// TIA Portal V20 export
FUNCTION_BLOCK "CallEquipment"   // FB25, LAD
TITLE = CallEquipment
// Template of an equipment module. This block contains the logic and futher calls (e.g. sequences, control modules, diagnostics etc.) of the equipment module.
// It can be used out of the box but also adapted to your own needs.
// stored: IsIECCheckEnabled true, MemoryReserve 100, Namespace Unit1.Em6, SetENOAutomatically true
   VAR_INPUT
      ZoneOperationEnable { ExternalWritable := 'False'} : "LWONIK_typeSafetyZoneManualOperation";
      unitEnableControlInterfaces { ExternalWritable := 'False'} : "LAF_typeEnableControlInterfaces";
      commandExcute { ExternalWritable := 'False'} : Bool;
   END_VAR
   VAR_IN_OUT
      unitStatus : "LAF_typeUnitStatus";   // Current unit status o be used in this EM
      emFeedback : "LUC_typeEmFeedback";   // Feedback of the EM to the Unit
      unitAlarmDB : "LAF_typeAlarms";   // Summarized EM Alarms for the Unit
   END_VAR
   VAR
      instSequenceVisionUnit { ExternalWritable := 'False'} : "Unit1.Em6.Sequence_1_VisionUnit";
      instSequenceVisionController { ExternalWritable := 'False'} : "Unit1.Em6.Sequence_2_VisionController";
      instSequenceQrRead { ExternalWritable := 'False'} : "Unit1.Em6.Sequence_3_QrRead";
      instVisionUnitInitializedJob1 { ExternalWritable := 'False'} : "LAF_SelectJob";
      instVisionUnitVisionPosJob2 { ExternalWritable := 'False'} : "LAF_SelectJob";
      instVisionUnitHomePosJob3 { ExternalWritable := 'False'} : "LAF_SelectJob";
      instVisionFullAutoJob10 { ExternalWritable := 'False'} : "LAF_SelectJob";
      instVisionControllerInitializedJob1 { ExternalWritable := 'False'} : "LAF_SelectJob";
      instVisionControllerInspectionJob2 { ExternalWritable := 'False'} : "LAF_SelectJob";
      instQrReaderInitializedJob1 { ExternalWritable := 'False'} : "LAF_SelectJob";
      instQrReaderQrReadJob2 { ExternalWritable := 'False'} : "LAF_SelectJob";
      instCmVisionAxisZ { ExternalWritable := 'False'} : "LBC_Axis64Pos_TecPlcCn";
      instCmVisionPusherSupportUpDown { ExternalWritable := 'False'} : "LBC_TwoWayActuatorCn";
      instCmVisionTriggerSensor { ExternalWritable := 'False'} : "LBC_DigitalSignalCn";
      instCmQrReader { ExternalWritable := 'False'} : "LER_QRread_SRX300";
      instCmQrReadHandy { ExternalWritable := 'False'} : "LER_QRread_DM8700";
      instVision_XGX2000 { ExternalWritable := 'False'} : "LER_Vision_XGX2000";
      instVision_XGX2000_Conversion { ExternalWritable := 'False'} : "LER_Vision_XGX2000_Conversion";
      instVisionAxisZControlInterlockSummary { ExternalWritable := 'False'} : "LER_Axis64Pos_InterlockSummary";
      instServoTorqueCal_DR9 { ExternalWritable := 'False'} : "LER_ServoTorqueCal";
      instLDrv701ControlVisionAxisZ { ExternalWritable := 'False'} : "LDrvSafe_SinaTlg701Control";   // Drive Telegram Function Library
      instLDrv701StatusVisionAxisZ { ExternalWritable := 'False'} : "LDrvSafe_SinaTlg701Status";   // Drive Telegram Function Library
      statUnitStatus { ExternalWritable := 'False'} : "LAF_typeUnitStatus";   // Unit Status used in this EM
      statAllBrakeTest { ExternalWritable := 'False'} : "LER_typeBrakeTestUnitCommands";
      instManageAlarms { ExternalWritable := 'False'} : "LAF_ManageAlarms";
      instEventsPFE { S7_SetPoint := 'True'} : "Unit1.Em6.EventsPFE";
      statPulse { ExternalWritable := 'False'} : Array[0..99] of Bool;
      statTonTimer { ExternalWritable := 'False'} : Array[0..99] of TON_TIME;
      statTofTimer { ExternalWritable := 'False'} : Array[0..99] of TOF_TIME;
      statEnableManualCmds { ExternalWritable := 'False'} : Bool;
      statGaugeCheck { ExternalWritable := 'False'} : Struct
         Type1Complete : Bool;
         Type3Compete : Bool;
      END_STRUCT;
      statSafeStateCheck { ExternalWritable := 'False'} : Struct
         VisionUnit : Bool;
         VisionController : Bool;
         VisionQrReader : Bool;
      END_STRUCT;
      statBobinID : String[32];
      citi_Ptrig : Array[0..20] of Bool;
      citiTon : Array[0..20] of TON_TIME;
      citi : Time;
      citiTest : Array[0..20] of Bool;
      statDataIncrease : Int;
   END_VAR
   VAR_TEMP
      tempScInProduction : Bool;   // Mode Production and StateComplete
      tempScNoProduction : Bool;   // Mode Manual and StateComplete
   END_VAR
   VAR CONSTANT
      TO_DO_INSERT_PRECONDITIONS_HERE : Bool := TRUE;   // Template : Add em specific conditions here
      NO_JOB : DInt;   // No job
      TRUE : Bool := TRUE;
      FALSE : Bool := FALSE;
      INIT_POSITION_NUMBER : SInt := -1;
      MIN_POSITION_NUMBER : SInt;
   END_VAR
   VAR_TEMP   // added for the SCL form of the ladder/FBD networks
      _w1 : Bool;
      _w2 : Bool;
      _w3 : Bool;
      _w4 : Bool;
      _w5 : Bool;
      _w6 : Bool;
      _w7 : Bool;
      _w8 : Bool;
      _w9 : Bool;
      _w10 : Bool;
      _w11 : Bool;
      _w12 : Bool;
      _w13 : Bool;
      _w14 : Bool;
      _w15 : Bool;
   END_VAR
BEGIN

REGION Network 1: BLOCK INFO HEADER
   // (company) / (C) Copyright (year)
   // ---------------------------------------------------------------------------------
   // Title:                             (Title of this block)
   // Comment/Function: (that is implemented in the block)
   // Library/Family:           (that the source is dedicated to)
   // Author:                        (department / person in charge / contact)
   // Target System:          (test system with FW version)
   // Engineering:              TIA Portal (SW version)
   // Restrictions:               (OB types, etc.)
   // Requirements:           (hardware, technological package, etc.)
   // ---------------------------------------------------------------------------------
   // Change log table:
   // Version          | Date             | Signature      | Expert in charge  | Changes applied ------------------------|----------------------|-------------------------|--------------------------------|-----------------------
   // 001.000.000 | yyyy-mm-dd | 0x00000000 | (name of expert) | First released version
END_REGION

REGION Network 2: DESCRIPTION
   // This is a template block provided by the Automation Framework. It can be used to create an own project.
   // The Block Info Header is prepared to put in your own data.
   // Description of the block could be added here and the docu created by Code2Docu.
END_REGION

REGION Network 3: ******************** Unit Input ********************
END_REGION

REGION Network 4: Em Nodes Brake Test
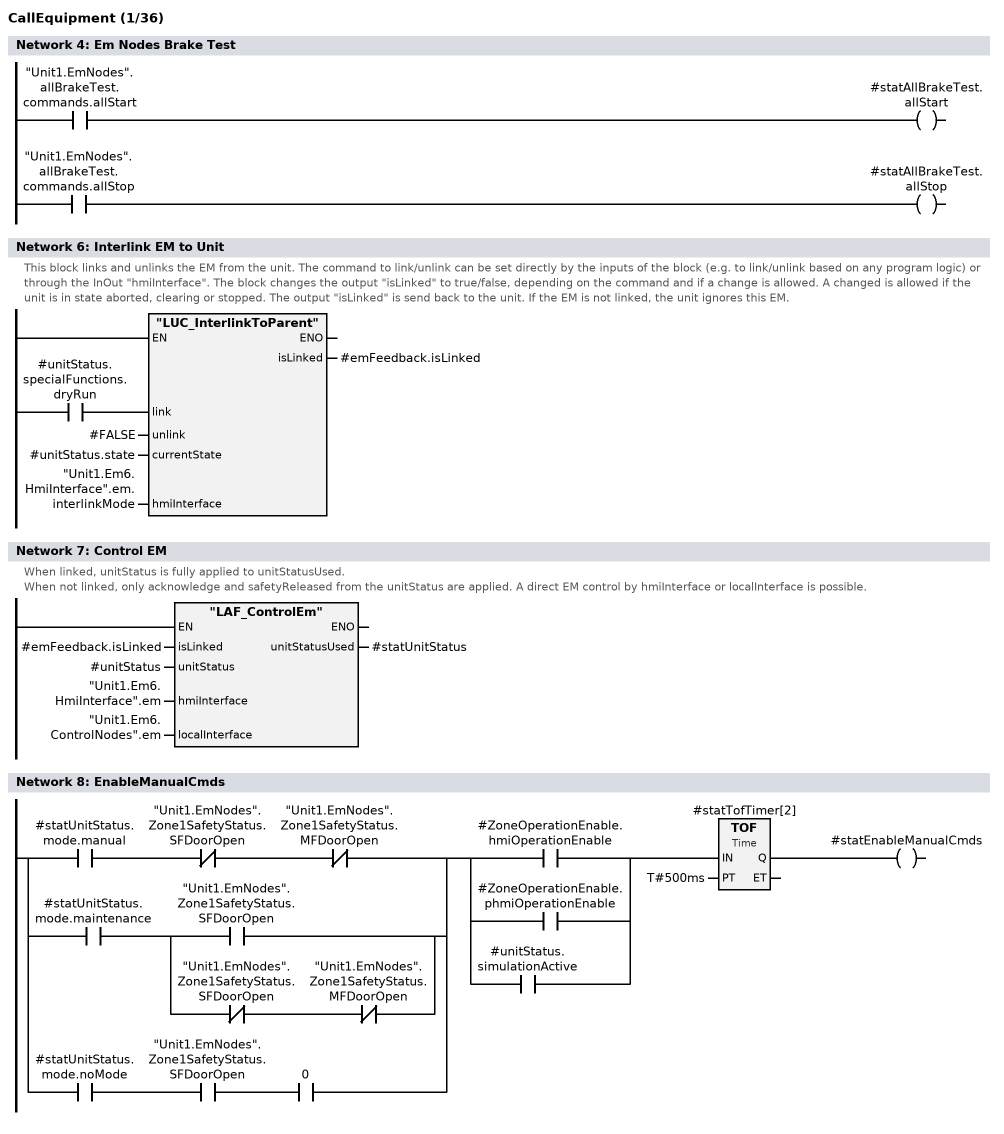
   RUNG wire#powerrail
      Contact( "Unit1.EmNodes".allBrakeTest.commands.allStart )
      Coil( #statAllBrakeTest.allStart )
   END_RUNG
   RUNG wire#powerrail
      Contact( "Unit1.EmNodes".allBrakeTest.commands.allStop )
      Coil( #statAllBrakeTest.allStop )
   END_RUNG
   // the same network as SCL:
   #statAllBrakeTest.allStart := "Unit1.EmNodes".allBrakeTest.commands.allStart;
   #statAllBrakeTest.allStop := "Unit1.EmNodes".allBrakeTest.commands.allStop;
END_REGION

REGION Network 5: ******************** Equipment Control ********************
END_REGION

REGION Network 6: Interlink EM to Unit
   // This block links and unlinks the EM from the unit. The command to link/unlink can be set directly by the inputs of the block (e.g. to link/unlink based on any program logic) or through the InOut "hmiInterface". The block changes the output "isLinked" to true/false, depending on the command and if a change is allowed. A changed is allowed if the unit is in state aborted, clearing or stopped. The output "isLinked" is send back to the unit. If the EM is not linked, the unit ignores this EM.
   RUNG wire#powerrail
      "LUC_InterlinkToParent"(link := wire#w1, unlink := #FALSE, currentState := #unitStatus.state, hmiInterface := "Unit1.Em6.HmiInterface".em.interlinkMode, isLinked => #emFeedback.isLinked)
   END_RUNG
   RUNG wire#powerrail
      Contact( #unitStatus.specialFunctions.dryRun )
   END_RUNG wire#w1
   // the same network as SCL:
   "LUC_InterlinkToParent"(link := #unitStatus.specialFunctions.dryRun,
                           unlink := #FALSE,
                           currentState := #unitStatus.state,
                           hmiInterface := "Unit1.Em6.HmiInterface".em.interlinkMode,
                           isLinked => #emFeedback.isLinked);
END_REGION

REGION Network 7: Control EM
   // When linked, unitStatus is fully applied to unitStatusUsed.
   // When not linked, only acknowledge and safetyReleased from the unitStatus are applied. A direct EM control by hmiInterface or localInterface is possible.
   RUNG wire#powerrail
      "LAF_ControlEm"(isLinked := #emFeedback.isLinked, unitStatus := #unitStatus, hmiInterface := "Unit1.Em6.HmiInterface".em, localInterface := "Unit1.Em6.ControlNodes".em, unitStatusUsed => #statUnitStatus)
   END_RUNG
   // the same network as SCL:
   "LAF_ControlEm"(isLinked := #emFeedback.isLinked,
                   unitStatus := #unitStatus,
                   hmiInterface := "Unit1.Em6.HmiInterface".em,
                   localInterface := "Unit1.Em6.ControlNodes".em,
                   unitStatusUsed => #statUnitStatus);
END_REGION

REGION Network 8: EnableManualCmds
   RUNG wire#powerrail
      Contact( #statUnitStatus.mode.manual )
      I_Contact( "Unit1.EmNodes".Zone1SafetyStatus.SFDoorOpen )
      I_Contact( "Unit1.EmNodes".Zone1SafetyStatus.MFDoorOpen )
      wire#w1
      Contact( #ZoneOperationEnable.hmiOperationEnable )
      wire#w3
      { S7_Templates := "time_type := Time" } #statTofTimer[2].TOF(pt := T#500ms, et =>)
      Coil( #statEnableManualCmds )
   END_RUNG
   RUNG wire#powerrail
      Contact( #statUnitStatus.mode.maintenance )
      wire#w2
      Contact( "Unit1.EmNodes".Zone1SafetyStatus.SFDoorOpen )
   END_RUNG wire#w1
   RUNG wire#w2
      I_Contact( "Unit1.EmNodes".Zone1SafetyStatus.SFDoorOpen )
      I_Contact( "Unit1.EmNodes".Zone1SafetyStatus.MFDoorOpen )
   END_RUNG wire#w1
   RUNG wire#powerrail
      Contact( #statUnitStatus.mode.noMode )
      Contact( "Unit1.EmNodes".Zone1SafetyStatus.SFDoorOpen )
      Contact( 0 )
   END_RUNG wire#w1
   RUNG wire#w1
      Contact( #ZoneOperationEnable.phmiOperationEnable )
   END_RUNG wire#w3
   RUNG wire#w1
      Contact( #unitStatus.simulationActive )
   END_RUNG wire#w3
   // the same network as SCL:
   #statTofTimer[2].TOF(IN := ((#statUnitStatus.mode.manual AND NOT "Unit1.EmNodes".Zone1SafetyStatus.SFDoorOpen AND NOT "Unit1.EmNodes".Zone1SafetyStatus.MFDoorOpen) OR (#statUnitStatus.mode.maintenance AND ("Unit1.EmNodes".Zone1SafetyStatus.SFDoorOpen OR (NOT "Unit1.EmNodes".Zone1SafetyStatus.SFDoorOpen AND NOT "Unit1.EmNodes".Zone1SafetyStatus.MFDoorOpen))) OR (#statUnitStatus.mode.noMode AND "Unit1.EmNodes".Zone1SafetyStatus.SFDoorOpen AND 0)) AND (#ZoneOperationEnable.hmiOperationEnable OR #ZoneOperationEnable.phmiOperationEnable OR #unitStatus.simulationActive),
                        PT := T#500ms);
   #statEnableManualCmds := #statTofTimer[2].Q;
END_REGION

REGION Network 9: Alarms Disabled
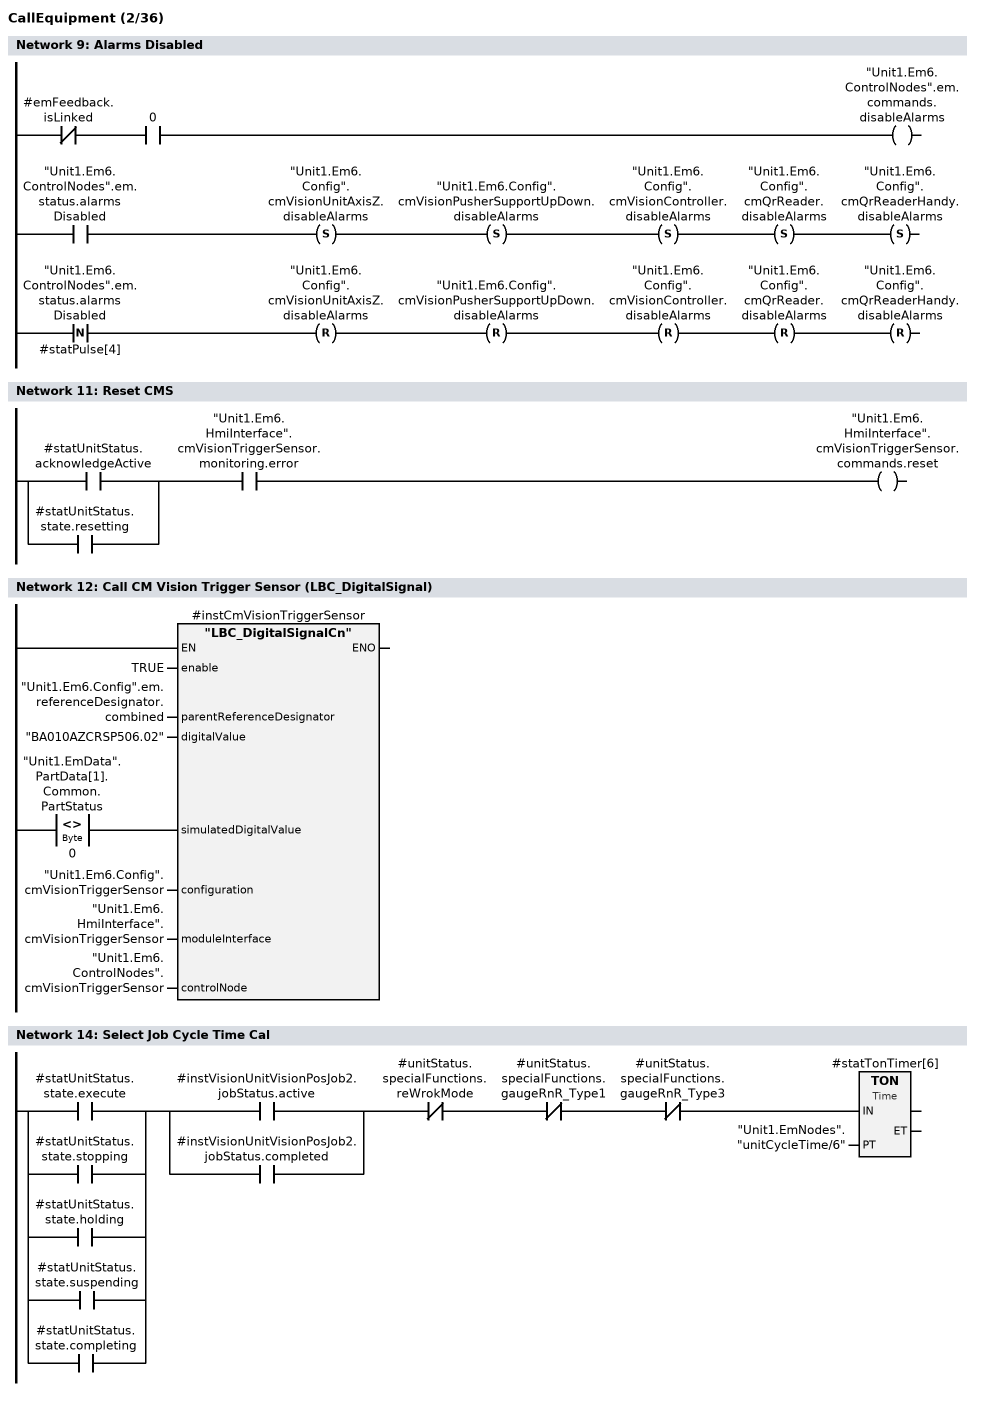
   RUNG wire#powerrail
      I_Contact( #emFeedback.isLinked )
      Contact( 0 )
      Coil( "Unit1.Em6.ControlNodes".em.commands.disableAlarms )
   END_RUNG
   RUNG wire#powerrail
      Contact( "Unit1.Em6.ControlNodes".em.status.alarmsDisabled )
      S_Coil( "Unit1.Em6.Config".cmVisionUnitAxisZ.disableAlarms )
      S_Coil( "Unit1.Em6.Config".cmVisionPusherSupportUpDown.disableAlarms )
      S_Coil( "Unit1.Em6.Config".cmVisionController.disableAlarms )
      S_Coil( "Unit1.Em6.Config".cmQrReader.disableAlarms )
      S_Coil( "Unit1.Em6.Config".cmQrReaderHandy.disableAlarms )
   END_RUNG
   RUNG wire#powerrail
      N_Contact(operand := "Unit1.Em6.ControlNodes".em.status.alarmsDisabled, bit := #statPulse[4])
      R_Coil( "Unit1.Em6.Config".cmVisionUnitAxisZ.disableAlarms )
      R_Coil( "Unit1.Em6.Config".cmVisionPusherSupportUpDown.disableAlarms )
      R_Coil( "Unit1.Em6.Config".cmVisionController.disableAlarms )
      R_Coil( "Unit1.Em6.Config".cmQrReader.disableAlarms )
      R_Coil( "Unit1.Em6.Config".cmQrReaderHandy.disableAlarms )
   END_RUNG
   // the same network as SCL:
   "Unit1.Em6.ControlNodes".em.commands.disableAlarms := NOT #emFeedback.isLinked AND 0;
   IF "Unit1.Em6.ControlNodes".em.status.alarmsDisabled THEN
       "Unit1.Em6.Config".cmVisionUnitAxisZ.disableAlarms := TRUE;
       "Unit1.Em6.Config".cmVisionPusherSupportUpDown.disableAlarms := TRUE;
       "Unit1.Em6.Config".cmVisionController.disableAlarms := TRUE;
       "Unit1.Em6.Config".cmQrReader.disableAlarms := TRUE;
       "Unit1.Em6.Config".cmQrReaderHandy.disableAlarms := TRUE;
   END_IF;
   #_w1 := NOT "Unit1.Em6.ControlNodes".em.status.alarmsDisabled AND #statPulse[4];   // falling edge of "Unit1.Em6.ControlNodes".em.status.alarmsDisabled
   #statPulse[4] := "Unit1.Em6.ControlNodes".em.status.alarmsDisabled;
   IF #_w1 THEN
       "Unit1.Em6.Config".cmVisionUnitAxisZ.disableAlarms := FALSE;
       "Unit1.Em6.Config".cmVisionPusherSupportUpDown.disableAlarms := FALSE;
       "Unit1.Em6.Config".cmVisionController.disableAlarms := FALSE;
       "Unit1.Em6.Config".cmQrReader.disableAlarms := FALSE;
       "Unit1.Em6.Config".cmQrReaderHandy.disableAlarms := FALSE;
   END_IF;
END_REGION

REGION Network 10: ******************** Control Modules (Sensors) ********************
   // Call control modules that are sensors before the em logic (jobs and sequence), so that the latest value is used in the logic.
END_REGION

REGION Network 11: Reset CMS
   RUNG wire#powerrail
      Contact( #statUnitStatus.acknowledgeActive )
      wire#w1
      Contact( "Unit1.Em6.HmiInterface".cmVisionTriggerSensor.monitoring.error )
      Coil( "Unit1.Em6.HmiInterface".cmVisionTriggerSensor.commands.reset )
   END_RUNG
   RUNG wire#powerrail
      Contact( #statUnitStatus.state.resetting )
   END_RUNG wire#w1
   // the same network as SCL:
   "Unit1.Em6.HmiInterface".cmVisionTriggerSensor.commands.reset := (#statUnitStatus.acknowledgeActive OR #statUnitStatus.state.resetting) AND "Unit1.Em6.HmiInterface".cmVisionTriggerSensor.monitoring.error;
END_REGION

REGION Network 12: Call CM Vision Trigger Sensor (LBC_DigitalSignal)
   RUNG wire#powerrail
      #instCmVisionTriggerSensor(simulatedDigitalValue := wire#w1, enable := TRUE, parentReferenceDesignator := "Unit1.Em6.Config".em.referenceDesignator.combined, digitalValue := "BA010AZCRSP506.02", configuration := "Unit1.Em6.Config".cmVisionTriggerSensor, moduleInterface := "Unit1.Em6.HmiInterface".cmVisionTriggerSensor, controlNode := "Unit1.Em6.ControlNodes".cmVisionTriggerSensor)
   END_RUNG
   RUNG wire#powerrail
      { S7_Templates := "SrcType := Byte" } NE_Contact(in1 := "Unit1.EmData".PartData[1].Common.PartStatus, in2 := 0)
   END_RUNG wire#w1
   // the same network as SCL:
   #instCmVisionTriggerSensor(enable := TRUE,   // "LBC_DigitalSignalCn"
                           parentReferenceDesignator := "Unit1.Em6.Config".em.referenceDesignator.combined,
                           digitalValue := "BA010AZCRSP506.02",
                           simulatedDigitalValue := "Unit1.EmData".PartData[1].Common.PartStatus <> 0,
                           configuration := "Unit1.Em6.Config".cmVisionTriggerSensor,
                           moduleInterface := "Unit1.Em6.HmiInterface".cmVisionTriggerSensor,
                           controlNode := "Unit1.Em6.ControlNodes".cmVisionTriggerSensor);
END_REGION

REGION Network 13: ******************** Equipment Logic ********************
END_REGION

REGION Network 14: Select Job Cycle Time Cal
   RUNG wire#powerrail
      Contact( #statUnitStatus.state.execute )
      wire#w1
      Contact( #instVisionUnitVisionPosJob2.jobStatus.active )
      wire#w2
      I_Contact( #unitStatus.specialFunctions.reWrokMode )
      I_Contact( #unitStatus.specialFunctions.gaugeRnR_Type1 )
      I_Contact( #unitStatus.specialFunctions.gaugeRnR_Type3 )
      { S7_Templates := "time_type := Time" } #statTonTimer[6].TON(pt := "Unit1.EmNodes"."unitCycleTime/6", et =>)
   END_RUNG
   RUNG wire#powerrail
      Contact( #statUnitStatus.state.stopping )
   END_RUNG wire#w1
   RUNG wire#powerrail
      Contact( #statUnitStatus.state.holding )
   END_RUNG wire#w1
   RUNG wire#powerrail
      Contact( #statUnitStatus.state.suspending )
   END_RUNG wire#w1
   RUNG wire#powerrail
      Contact( #statUnitStatus.state.completing )
   END_RUNG wire#w1
   RUNG wire#w1
      Contact( #instVisionUnitVisionPosJob2.jobStatus.completed )
   END_RUNG wire#w2
   // the same network as SCL:
   #statTonTimer[6].TON(IN := (#statUnitStatus.state.execute OR #statUnitStatus.state.stopping OR #statUnitStatus.state.holding OR #statUnitStatus.state.suspending OR #statUnitStatus.state.completing) AND (#instVisionUnitVisionPosJob2.jobStatus.active OR #instVisionUnitVisionPosJob2.jobStatus.completed) AND NOT #unitStatus.specialFunctions.reWrokMode AND NOT #unitStatus.specialFunctions.gaugeRnR_Type1 AND NOT #unitStatus.specialFunctions.gaugeRnR_Type3,
                        PT := "Unit1.EmNodes"."unitCycleTime/6");
END_REGION

REGION Network 15: Map Unit Status to Sequence Status [1] Vision Unit
   // This block maps the unit status to the seuqnce status. Thus, it controls the sequence depending on the unit status. E.g. it sets the sequence to automatic when the unit state is in productions. This blocks work perfectly with the sequences provided in the AF. 
   // This typed block (MapUnitStatusToSequence) could be adjusted to specific application requirements or if other, user-defined sequences are used.
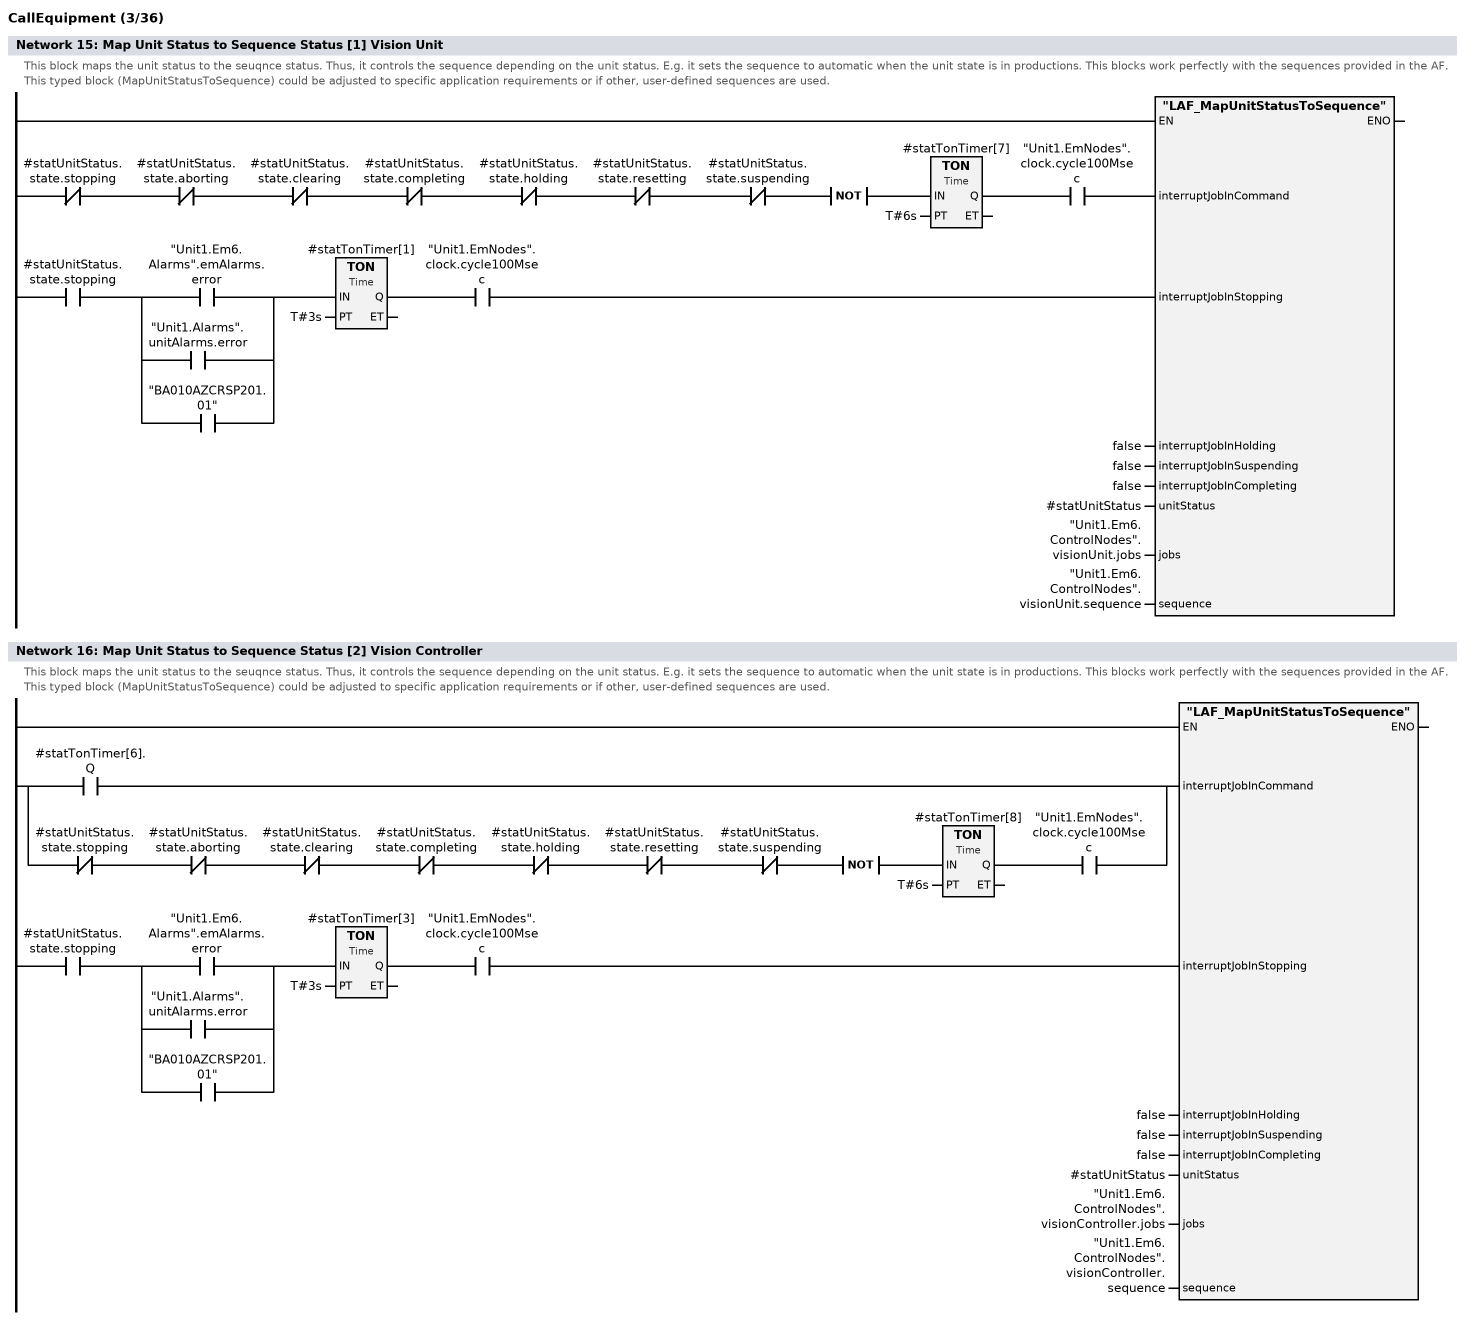
   RUNG wire#powerrail
      "LAF_MapUnitStatusToSequence"(interruptJobInCommand := wire#w1, interruptJobInStopping := wire#w4, interruptJobInHolding := false, interruptJobInSuspending := false, interruptJobInCompleting := false, unitStatus := #statUnitStatus, jobs := "Unit1.Em6.ControlNodes".visionUnit.jobs, sequence := "Unit1.Em6.ControlNodes".visionUnit.sequence)
   END_RUNG
   RUNG wire#powerrail
      I_Contact( #statUnitStatus.state.stopping )
      I_Contact( #statUnitStatus.state.aborting )
      I_Contact( #statUnitStatus.state.clearing )
      I_Contact( #statUnitStatus.state.completing )
      I_Contact( #statUnitStatus.state.holding )
      I_Contact( #statUnitStatus.state.resetting )
      I_Contact( #statUnitStatus.state.suspending )
      Not()
      { S7_Templates := "time_type := Time" } #statTonTimer[7].TON(pt := T#6s, et =>)
      Contact( "Unit1.EmNodes".clock.cycle100Msec )
   END_RUNG wire#w1
   RUNG wire#powerrail
      Contact( #statUnitStatus.state.stopping )
      wire#w2
      Contact( "Unit1.Em6.Alarms".emAlarms.error )
      wire#w3
      { S7_Templates := "time_type := Time" } #statTonTimer[1].TON(pt := T#3s, et =>)
      Contact( "Unit1.EmNodes".clock.cycle100Msec )
   END_RUNG wire#w4
   RUNG wire#w2
      Contact( "Unit1.Alarms".unitAlarms.error )
   END_RUNG wire#w3
   RUNG wire#w2
      Contact( "BA010AZCRSP201.01" )
   END_RUNG wire#w3
   // the same network as SCL:
   #statTonTimer[7].TON(IN := NOT (NOT #statUnitStatus.state.stopping AND NOT #statUnitStatus.state.aborting AND NOT #statUnitStatus.state.clearing AND NOT #statUnitStatus.state.completing AND NOT #statUnitStatus.state.holding AND NOT #statUnitStatus.state.resetting AND NOT #statUnitStatus.state.suspending),
                        PT := T#6s);
   #_w1 := #statTonTimer[7].Q AND "Unit1.EmNodes".clock.cycle100Msec;
   #statTonTimer[1].TON(IN := #statUnitStatus.state.stopping AND ("Unit1.Em6.Alarms".emAlarms.error OR "Unit1.Alarms".unitAlarms.error OR "BA010AZCRSP201.01"),
                        PT := T#3s);
   "LAF_MapUnitStatusToSequence"(interruptJobInCommand := #_w1,
                           interruptJobInStopping := #statTonTimer[1].Q AND "Unit1.EmNodes".clock.cycle100Msec,
                           interruptJobInHolding := false,
                           interruptJobInSuspending := false,
                           interruptJobInCompleting := false,
                           unitStatus := #statUnitStatus,
                           jobs := "Unit1.Em6.ControlNodes".visionUnit.jobs,
                           sequence := "Unit1.Em6.ControlNodes".visionUnit.sequence);
END_REGION

REGION Network 16: Map Unit Status to Sequence Status [2] Vision Controller
   // This block maps the unit status to the seuqnce status. Thus, it controls the sequence depending on the unit status. E.g. it sets the sequence to automatic when the unit state is in productions. This blocks work perfectly with the sequences provided in the AF. 
   // This typed block (MapUnitStatusToSequence) could be adjusted to specific application requirements or if other, user-defined sequences are used.
   RUNG wire#powerrail
      "LAF_MapUnitStatusToSequence"(interruptJobInCommand := wire#w1, interruptJobInStopping := wire#w4, interruptJobInHolding := false, interruptJobInSuspending := false, interruptJobInCompleting := false, unitStatus := #statUnitStatus, jobs := "Unit1.Em6.ControlNodes".visionController.jobs, sequence := "Unit1.Em6.ControlNodes".visionController.sequence)
   END_RUNG
   RUNG wire#powerrail
      Contact( #statTonTimer[6].Q )
   END_RUNG wire#w1
   RUNG wire#powerrail
      I_Contact( #statUnitStatus.state.stopping )
      I_Contact( #statUnitStatus.state.aborting )
      I_Contact( #statUnitStatus.state.clearing )
      I_Contact( #statUnitStatus.state.completing )
      I_Contact( #statUnitStatus.state.holding )
      I_Contact( #statUnitStatus.state.resetting )
      I_Contact( #statUnitStatus.state.suspending )
      Not()
      { S7_Templates := "time_type := Time" } #statTonTimer[8].TON(pt := T#6s, et =>)
      Contact( "Unit1.EmNodes".clock.cycle100Msec )
   END_RUNG wire#w1
   RUNG wire#powerrail
      Contact( #statUnitStatus.state.stopping )
      wire#w2
      Contact( "Unit1.Em6.Alarms".emAlarms.error )
      wire#w3
      { S7_Templates := "time_type := Time" } #statTonTimer[3].TON(pt := T#3s, et =>)
      Contact( "Unit1.EmNodes".clock.cycle100Msec )
   END_RUNG wire#w4
   RUNG wire#w2
      Contact( "Unit1.Alarms".unitAlarms.error )
   END_RUNG wire#w3
   RUNG wire#w2
      Contact( "BA010AZCRSP201.01" )
   END_RUNG wire#w3
   // the same network as SCL:
   #_w1 := #statTonTimer[6].Q;
   #statTonTimer[8].TON(IN := NOT (NOT #statUnitStatus.state.stopping AND NOT #statUnitStatus.state.aborting AND NOT #statUnitStatus.state.clearing AND NOT #statUnitStatus.state.completing AND NOT #statUnitStatus.state.holding AND NOT #statUnitStatus.state.resetting AND NOT #statUnitStatus.state.suspending),
                        PT := T#6s);
   #_w2 := #_w1 OR (#statTonTimer[8].Q AND "Unit1.EmNodes".clock.cycle100Msec);
   #statTonTimer[3].TON(IN := #statUnitStatus.state.stopping AND ("Unit1.Em6.Alarms".emAlarms.error OR "Unit1.Alarms".unitAlarms.error OR "BA010AZCRSP201.01"),
                        PT := T#3s);
   "LAF_MapUnitStatusToSequence"(interruptJobInCommand := #_w2,
                           interruptJobInStopping := #statTonTimer[3].Q AND "Unit1.EmNodes".clock.cycle100Msec,
                           interruptJobInHolding := false,
                           interruptJobInSuspending := false,
                           interruptJobInCompleting := false,
                           unitStatus := #statUnitStatus,
                           jobs := "Unit1.Em6.ControlNodes".visionController.jobs,
                           sequence := "Unit1.Em6.ControlNodes".visionController.sequence);
END_REGION

REGION Network 17: Map Unit Status to Sequence Status [3] QrRead
   // This block maps the unit status to the seuqnce status. Thus, it controls the sequence depending on the unit status. E.g. it sets the sequence to automatic when the unit state is in productions. This blocks work perfectly with the sequences provided in the AF. 
   // This typed block (MapUnitStatusToSequence) could be adjusted to specific application requirements or if other, user-defined sequences are used.
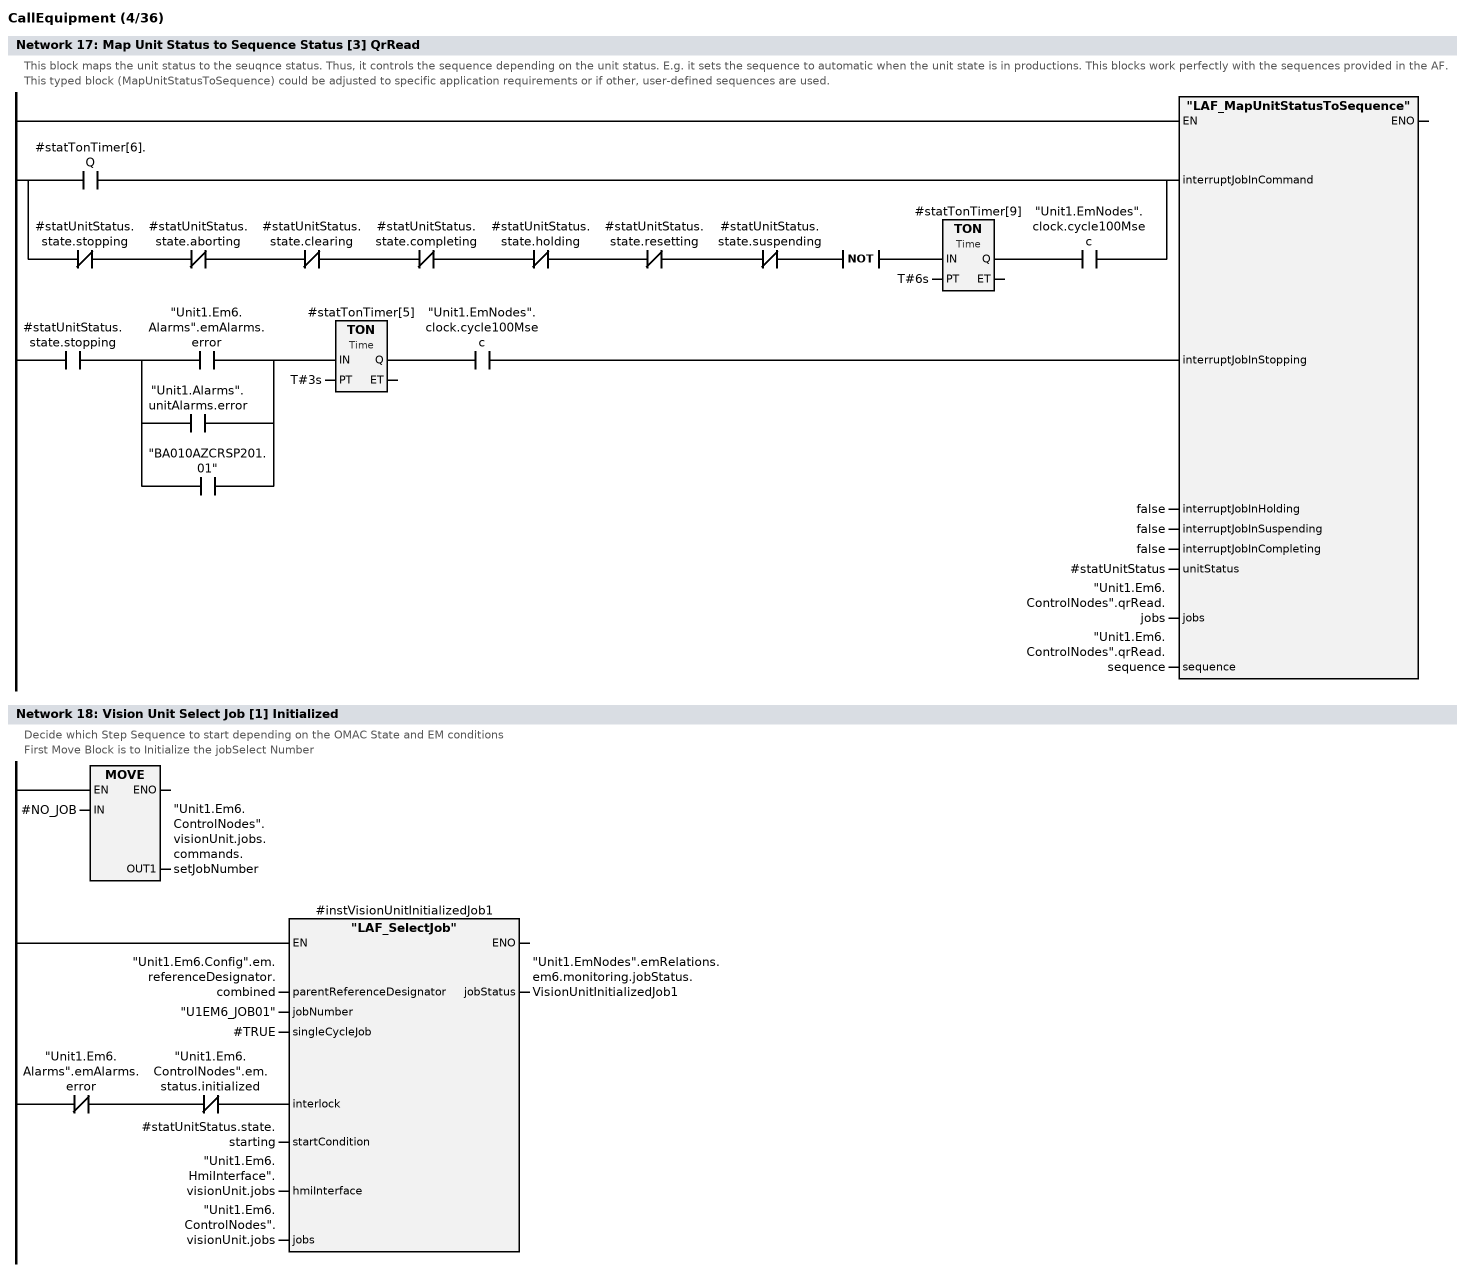
   RUNG wire#powerrail
      "LAF_MapUnitStatusToSequence"(interruptJobInCommand := wire#w1, interruptJobInStopping := wire#w4, interruptJobInHolding := false, interruptJobInSuspending := false, interruptJobInCompleting := false, unitStatus := #statUnitStatus, jobs := "Unit1.Em6.ControlNodes".qrRead.jobs, sequence := "Unit1.Em6.ControlNodes".qrRead.sequence)
   END_RUNG
   RUNG wire#powerrail
      Contact( #statTonTimer[6].Q )
   END_RUNG wire#w1
   RUNG wire#powerrail
      I_Contact( #statUnitStatus.state.stopping )
      I_Contact( #statUnitStatus.state.aborting )
      I_Contact( #statUnitStatus.state.clearing )
      I_Contact( #statUnitStatus.state.completing )
      I_Contact( #statUnitStatus.state.holding )
      I_Contact( #statUnitStatus.state.resetting )
      I_Contact( #statUnitStatus.state.suspending )
      Not()
      { S7_Templates := "time_type := Time" } #statTonTimer[9].TON(pt := T#6s, et =>)
      Contact( "Unit1.EmNodes".clock.cycle100Msec )
   END_RUNG wire#w1
   RUNG wire#powerrail
      Contact( #statUnitStatus.state.stopping )
      wire#w2
      Contact( "Unit1.Em6.Alarms".emAlarms.error )
      wire#w3
      { S7_Templates := "time_type := Time" } #statTonTimer[5].TON(pt := T#3s, et =>)
      Contact( "Unit1.EmNodes".clock.cycle100Msec )
   END_RUNG wire#w4
   RUNG wire#w2
      Contact( "Unit1.Alarms".unitAlarms.error )
   END_RUNG wire#w3
   RUNG wire#w2
      Contact( "BA010AZCRSP201.01" )
   END_RUNG wire#w3
   // the same network as SCL:
   #_w1 := #statTonTimer[6].Q;
   #statTonTimer[9].TON(IN := NOT (NOT #statUnitStatus.state.stopping AND NOT #statUnitStatus.state.aborting AND NOT #statUnitStatus.state.clearing AND NOT #statUnitStatus.state.completing AND NOT #statUnitStatus.state.holding AND NOT #statUnitStatus.state.resetting AND NOT #statUnitStatus.state.suspending),
                        PT := T#6s);
   #_w2 := #_w1 OR (#statTonTimer[9].Q AND "Unit1.EmNodes".clock.cycle100Msec);
   #statTonTimer[5].TON(IN := #statUnitStatus.state.stopping AND ("Unit1.Em6.Alarms".emAlarms.error OR "Unit1.Alarms".unitAlarms.error OR "BA010AZCRSP201.01"),
                        PT := T#3s);
   "LAF_MapUnitStatusToSequence"(interruptJobInCommand := #_w2,
                           interruptJobInStopping := #statTonTimer[5].Q AND "Unit1.EmNodes".clock.cycle100Msec,
                           interruptJobInHolding := false,
                           interruptJobInSuspending := false,
                           interruptJobInCompleting := false,
                           unitStatus := #statUnitStatus,
                           jobs := "Unit1.Em6.ControlNodes".qrRead.jobs,
                           sequence := "Unit1.Em6.ControlNodes".qrRead.sequence);
END_REGION

REGION Network 18: Vision Unit Select Job [1] Initialized
   // Decide which Step Sequence to start depending on the OMAC State and EM conditions
   // First Move Block is to Initialize the jobSelect Number
   RUNG wire#powerrail
      Move(in := #NO_JOB, out1 => "Unit1.Em6.ControlNodes".visionUnit.jobs.commands.setJobNumber)
   END_RUNG
   RUNG wire#powerrail
      #instVisionUnitInitializedJob1(interlock := wire#w1, parentReferenceDesignator := "Unit1.Em6.Config".em.referenceDesignator.combined, jobNumber := "U1EM6_JOB01", singleCycleJob := #TRUE, startCondition := #statUnitStatus.state.starting, hmiInterface := "Unit1.Em6.HmiInterface".visionUnit.jobs, jobs := "Unit1.Em6.ControlNodes".visionUnit.jobs, jobStatus => "Unit1.EmNodes".emRelations.em6.monitoring.jobStatus.VisionUnitInitializedJob1)
   END_RUNG
   RUNG wire#powerrail
      I_Contact( "Unit1.Em6.Alarms".emAlarms.error )
      I_Contact( "Unit1.Em6.ControlNodes".em.status.initialized )
   END_RUNG wire#w1
   // the same network as SCL:
   "Unit1.Em6.ControlNodes".visionUnit.jobs.commands.setJobNumber := #NO_JOB;
   #instVisionUnitInitializedJob1(parentReferenceDesignator := "Unit1.Em6.Config".em.referenceDesignator.combined,   // "LAF_SelectJob"
                           jobNumber := "U1EM6_JOB01",
                           singleCycleJob := #TRUE,
                           interlock := NOT "Unit1.Em6.Alarms".emAlarms.error AND NOT "Unit1.Em6.ControlNodes".em.status.initialized,
                           startCondition := #statUnitStatus.state.starting,
                           hmiInterface := "Unit1.Em6.HmiInterface".visionUnit.jobs,
                           jobs := "Unit1.Em6.ControlNodes".visionUnit.jobs,
                           jobStatus => "Unit1.EmNodes".emRelations.em6.monitoring.jobStatus.VisionUnitInitializedJob1);
END_REGION

REGION Network 19: Vision Unit Select Job [2] VisionPos Auto
   // Decide which Step Sequence to start depending on the OMAC State and EM conditions
   // First Move Block is to Initialize the jobSelect Number
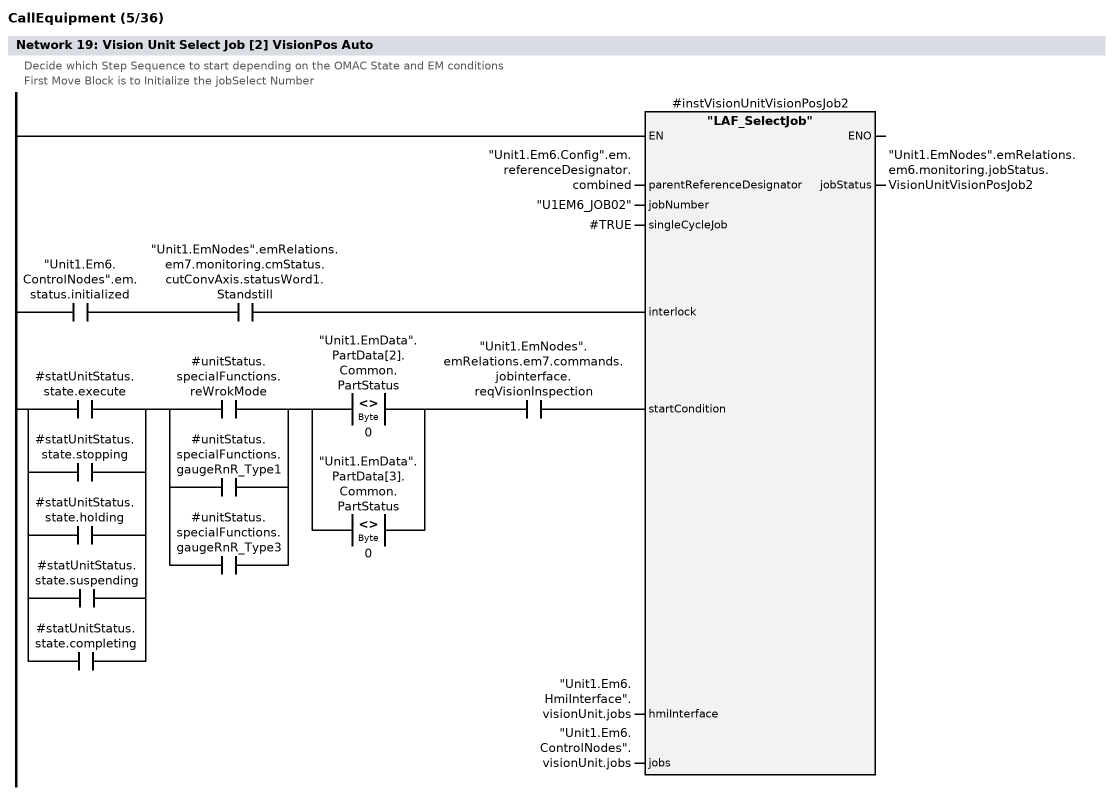
   RUNG wire#powerrail
      #instVisionUnitVisionPosJob2(interlock := wire#w1, startCondition := wire#w5, parentReferenceDesignator := "Unit1.Em6.Config".em.referenceDesignator.combined, jobNumber := "U1EM6_JOB02", singleCycleJob := #TRUE, hmiInterface := "Unit1.Em6.HmiInterface".visionUnit.jobs, jobs := "Unit1.Em6.ControlNodes".visionUnit.jobs, jobStatus => "Unit1.EmNodes".emRelations.em6.monitoring.jobStatus.VisionUnitVisionPosJob2)
   END_RUNG
   RUNG wire#powerrail
      Contact( "Unit1.Em6.ControlNodes".em.status.initialized )
      Contact( "Unit1.EmNodes".emRelations.em7.monitoring.cmStatus.cutConvAxis.statusWord1.Standstill )
   END_RUNG wire#w1
   RUNG wire#powerrail
      Contact( #statUnitStatus.state.execute )
      wire#w2
      Contact( #unitStatus.specialFunctions.reWrokMode )
      wire#w3
      { S7_Templates := "SrcType := Byte" } NE_Contact(in1 := "Unit1.EmData".PartData[2].Common.PartStatus, in2 := 0)
      wire#w4
      Contact( "Unit1.EmNodes".emRelations.em7.commands.jobinterface.reqVisionInspection )
   END_RUNG wire#w5
   RUNG wire#powerrail
      Contact( #statUnitStatus.state.stopping )
   END_RUNG wire#w2
   RUNG wire#powerrail
      Contact( #statUnitStatus.state.holding )
   END_RUNG wire#w2
   RUNG wire#powerrail
      Contact( #statUnitStatus.state.suspending )
   END_RUNG wire#w2
   RUNG wire#powerrail
      Contact( #statUnitStatus.state.completing )
   END_RUNG wire#w2
   RUNG wire#w2
      Contact( #unitStatus.specialFunctions.gaugeRnR_Type1 )
   END_RUNG wire#w3
   RUNG wire#w2
      Contact( #unitStatus.specialFunctions.gaugeRnR_Type3 )
   END_RUNG wire#w3
   RUNG wire#w3
      { S7_Templates := "SrcType := Byte" } NE_Contact(in1 := "Unit1.EmData".PartData[3].Common.PartStatus, in2 := 0)
   END_RUNG wire#w4
   // the same network as SCL:
   #instVisionUnitVisionPosJob2(parentReferenceDesignator := "Unit1.Em6.Config".em.referenceDesignator.combined,   // "LAF_SelectJob"
                           jobNumber := "U1EM6_JOB02",
                           singleCycleJob := #TRUE,
                           interlock := "Unit1.Em6.ControlNodes".em.status.initialized AND "Unit1.EmNodes".emRelations.em7.monitoring.cmStatus.cutConvAxis.statusWord1.Standstill,
                           startCondition := (#statUnitStatus.state.execute OR #statUnitStatus.state.stopping OR #statUnitStatus.state.holding OR #statUnitStatus.state.suspending OR #statUnitStatus.state.completing) AND (#unitStatus.specialFunctions.reWrokMode OR #unitStatus.specialFunctions.gaugeRnR_Type1 OR #unitStatus.specialFunctions.gaugeRnR_Type3) AND (("Unit1.EmData".PartData[2].Common.PartStatus <> 0) OR ("Unit1.EmData".PartData[3].Common.PartStatus <> 0)) AND "Unit1.EmNodes".emRelations.em7.commands.jobinterface.reqVisionInspection,
                           hmiInterface := "Unit1.Em6.HmiInterface".visionUnit.jobs,
                           jobs := "Unit1.Em6.ControlNodes".visionUnit.jobs,
                           jobStatus => "Unit1.EmNodes".emRelations.em6.monitoring.jobStatus.VisionUnitVisionPosJob2);
END_REGION

REGION Network 20: Vision Unit Select Job [3] HomePos Auto
   // Decide which Step Sequence to start depending on the OMAC State and EM conditions
   // First Move Block is to Initialize the jobSelect Number
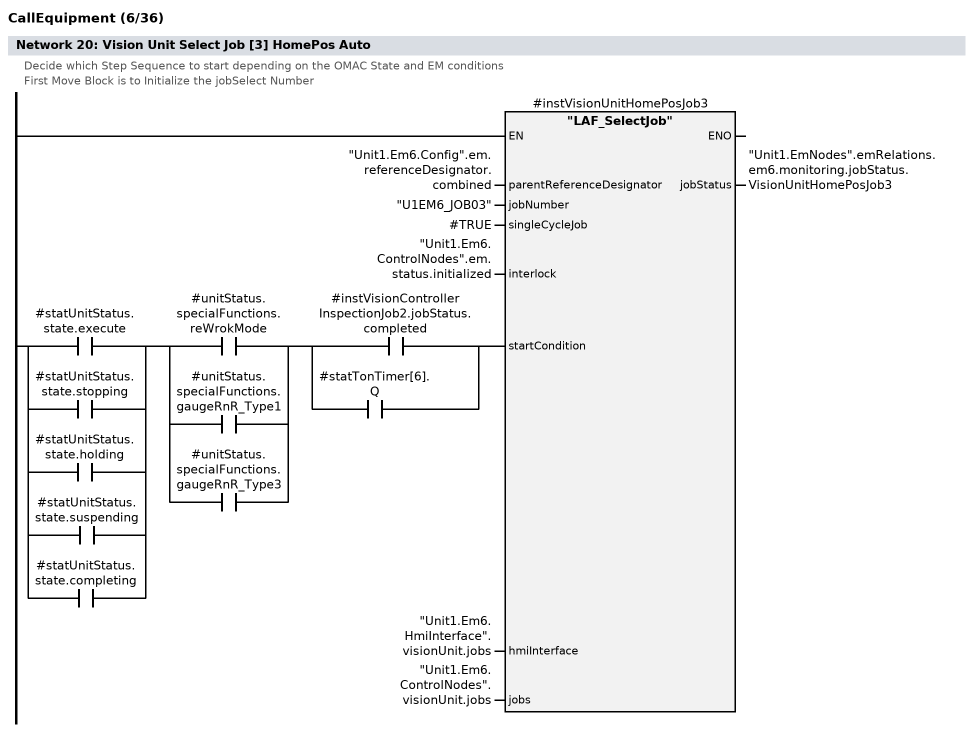
   RUNG wire#powerrail
      #instVisionUnitHomePosJob3(startCondition := wire#w3, parentReferenceDesignator := "Unit1.Em6.Config".em.referenceDesignator.combined, jobNumber := "U1EM6_JOB03", singleCycleJob := #TRUE, interlock := "Unit1.Em6.ControlNodes".em.status.initialized, hmiInterface := "Unit1.Em6.HmiInterface".visionUnit.jobs, jobs := "Unit1.Em6.ControlNodes".visionUnit.jobs, jobStatus => "Unit1.EmNodes".emRelations.em6.monitoring.jobStatus.VisionUnitHomePosJob3)
   END_RUNG
   RUNG wire#powerrail
      Contact( #statUnitStatus.state.execute )
      wire#w1
      Contact( #unitStatus.specialFunctions.reWrokMode )
      wire#w2
      Contact( #instVisionControllerInspectionJob2.jobStatus.completed )
   END_RUNG wire#w3
   RUNG wire#powerrail
      Contact( #statUnitStatus.state.stopping )
   END_RUNG wire#w1
   RUNG wire#powerrail
      Contact( #statUnitStatus.state.holding )
   END_RUNG wire#w1
   RUNG wire#powerrail
      Contact( #statUnitStatus.state.suspending )
   END_RUNG wire#w1
   RUNG wire#powerrail
      Contact( #statUnitStatus.state.completing )
   END_RUNG wire#w1
   RUNG wire#w1
      Contact( #unitStatus.specialFunctions.gaugeRnR_Type1 )
   END_RUNG wire#w2
   RUNG wire#w1
      Contact( #unitStatus.specialFunctions.gaugeRnR_Type3 )
   END_RUNG wire#w2
   RUNG wire#w2
      Contact( #statTonTimer[6].Q )
   END_RUNG wire#w3
   // the same network as SCL:
   #instVisionUnitHomePosJob3(parentReferenceDesignator := "Unit1.Em6.Config".em.referenceDesignator.combined,   // "LAF_SelectJob"
                           jobNumber := "U1EM6_JOB03",
                           singleCycleJob := #TRUE,
                           interlock := "Unit1.Em6.ControlNodes".em.status.initialized,
                           startCondition := (#statUnitStatus.state.execute OR #statUnitStatus.state.stopping OR #statUnitStatus.state.holding OR #statUnitStatus.state.suspending OR #statUnitStatus.state.completing) AND (#unitStatus.specialFunctions.reWrokMode OR #unitStatus.specialFunctions.gaugeRnR_Type1 OR #unitStatus.specialFunctions.gaugeRnR_Type3) AND (#instVisionControllerInspectionJob2.jobStatus.completed OR #statTonTimer[6].Q),
                           hmiInterface := "Unit1.Em6.HmiInterface".visionUnit.jobs,
                           jobs := "Unit1.Em6.ControlNodes".visionUnit.jobs,
                           jobStatus => "Unit1.EmNodes".emRelations.em6.monitoring.jobStatus.VisionUnitHomePosJob3);
END_REGION

REGION Network 21: Vision Unit Select Job [10] Vision Full Auto
   // Decide which Step Sequence to start depending on the OMAC State and EM conditions
   // First Move Block is to Initialize the jobSelect Number
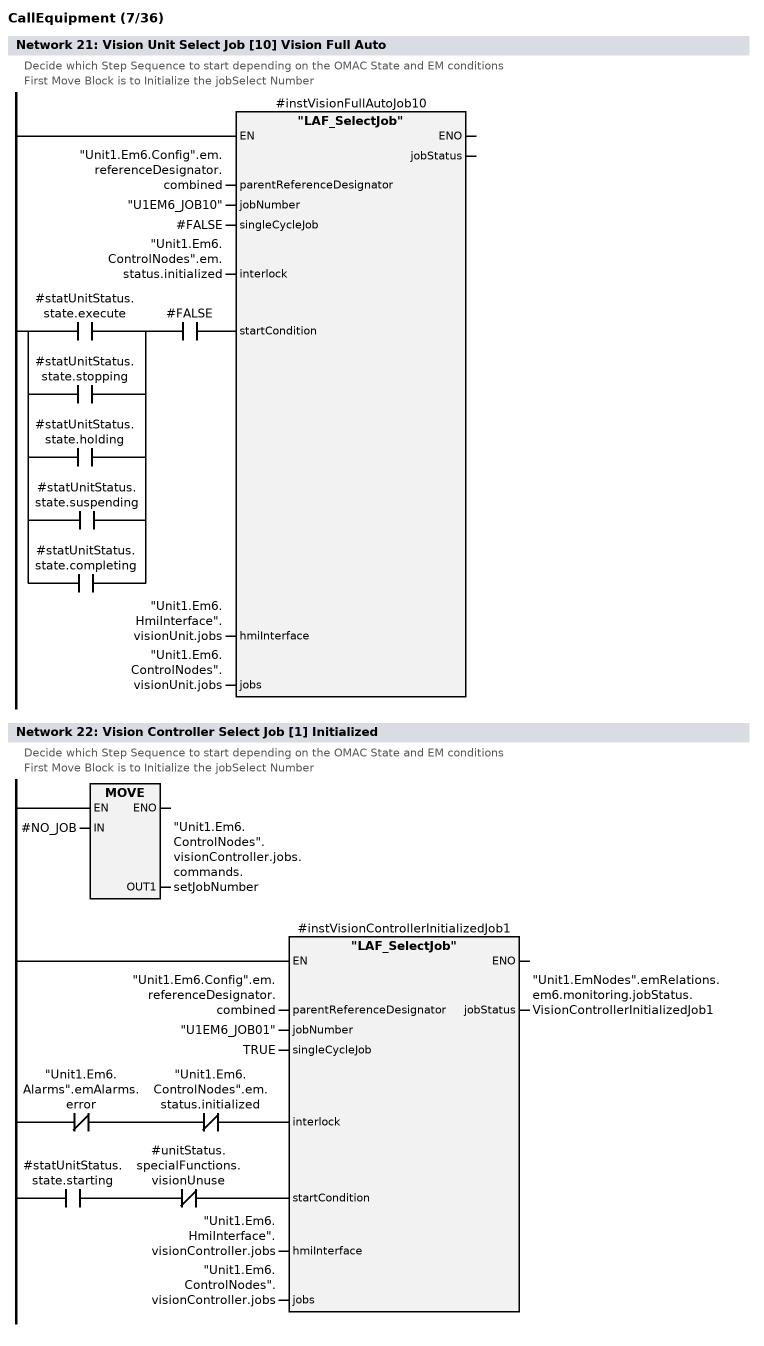
   RUNG wire#powerrail
      #instVisionFullAutoJob10(startCondition := wire#w2, parentReferenceDesignator := "Unit1.Em6.Config".em.referenceDesignator.combined, jobNumber := "U1EM6_JOB10", singleCycleJob := #FALSE, interlock := "Unit1.Em6.ControlNodes".em.status.initialized, hmiInterface := "Unit1.Em6.HmiInterface".visionUnit.jobs, jobs := "Unit1.Em6.ControlNodes".visionUnit.jobs, jobStatus =>)
   END_RUNG
   RUNG wire#powerrail
      Contact( #statUnitStatus.state.execute )
      wire#w1
      Contact( #FALSE )
   END_RUNG wire#w2
   RUNG wire#powerrail
      Contact( #statUnitStatus.state.stopping )
   END_RUNG wire#w1
   RUNG wire#powerrail
      Contact( #statUnitStatus.state.holding )
   END_RUNG wire#w1
   RUNG wire#powerrail
      Contact( #statUnitStatus.state.suspending )
   END_RUNG wire#w1
   RUNG wire#powerrail
      Contact( #statUnitStatus.state.completing )
   END_RUNG wire#w1
   // the same network as SCL:
   #instVisionFullAutoJob10(parentReferenceDesignator := "Unit1.Em6.Config".em.referenceDesignator.combined,   // "LAF_SelectJob"
                           jobNumber := "U1EM6_JOB10",
                           singleCycleJob := #FALSE,
                           interlock := "Unit1.Em6.ControlNodes".em.status.initialized,
                           startCondition := (#statUnitStatus.state.execute OR #statUnitStatus.state.stopping OR #statUnitStatus.state.holding OR #statUnitStatus.state.suspending OR #statUnitStatus.state.completing) AND #FALSE,
                           hmiInterface := "Unit1.Em6.HmiInterface".visionUnit.jobs,
                           jobs := "Unit1.Em6.ControlNodes".visionUnit.jobs);
END_REGION

REGION Network 22: Vision Controller Select Job [1] Initialized
   // Decide which Step Sequence to start depending on the OMAC State and EM conditions
   // First Move Block is to Initialize the jobSelect Number
   RUNG wire#powerrail
      Move(in := #NO_JOB, out1 => "Unit1.Em6.ControlNodes".visionController.jobs.commands.setJobNumber)
   END_RUNG
   RUNG wire#powerrail
      #instVisionControllerInitializedJob1(interlock := wire#w1, startCondition := wire#w2, parentReferenceDesignator := "Unit1.Em6.Config".em.referenceDesignator.combined, jobNumber := "U1EM6_JOB01", singleCycleJob := TRUE, hmiInterface := "Unit1.Em6.HmiInterface".visionController.jobs, jobs := "Unit1.Em6.ControlNodes".visionController.jobs, jobStatus => "Unit1.EmNodes".emRelations.em6.monitoring.jobStatus.VisionControllerInitializedJob1)
   END_RUNG
   RUNG wire#powerrail
      I_Contact( "Unit1.Em6.Alarms".emAlarms.error )
      I_Contact( "Unit1.Em6.ControlNodes".em.status.initialized )
   END_RUNG wire#w1
   RUNG wire#powerrail
      Contact( #statUnitStatus.state.starting )
      I_Contact( #unitStatus.specialFunctions.visionUnuse )
   END_RUNG wire#w2
   // the same network as SCL:
   "Unit1.Em6.ControlNodes".visionController.jobs.commands.setJobNumber := #NO_JOB;
   #instVisionControllerInitializedJob1(parentReferenceDesignator := "Unit1.Em6.Config".em.referenceDesignator.combined,   // "LAF_SelectJob"
                           jobNumber := "U1EM6_JOB01",
                           singleCycleJob := TRUE,
                           interlock := NOT "Unit1.Em6.Alarms".emAlarms.error AND NOT "Unit1.Em6.ControlNodes".em.status.initialized,
                           startCondition := #statUnitStatus.state.starting AND NOT #unitStatus.specialFunctions.visionUnuse,
                           hmiInterface := "Unit1.Em6.HmiInterface".visionController.jobs,
                           jobs := "Unit1.Em6.ControlNodes".visionController.jobs,
                           jobStatus => "Unit1.EmNodes".emRelations.em6.monitoring.jobStatus.VisionControllerInitializedJob1);
END_REGION

REGION Network 23: Vision Controller Select Job [2] Vision Inspection Auto
   // Decide which Step Sequence to start depending on the OMAC State and EM conditions
   // First Move Block is to Initialize the jobSelect Number
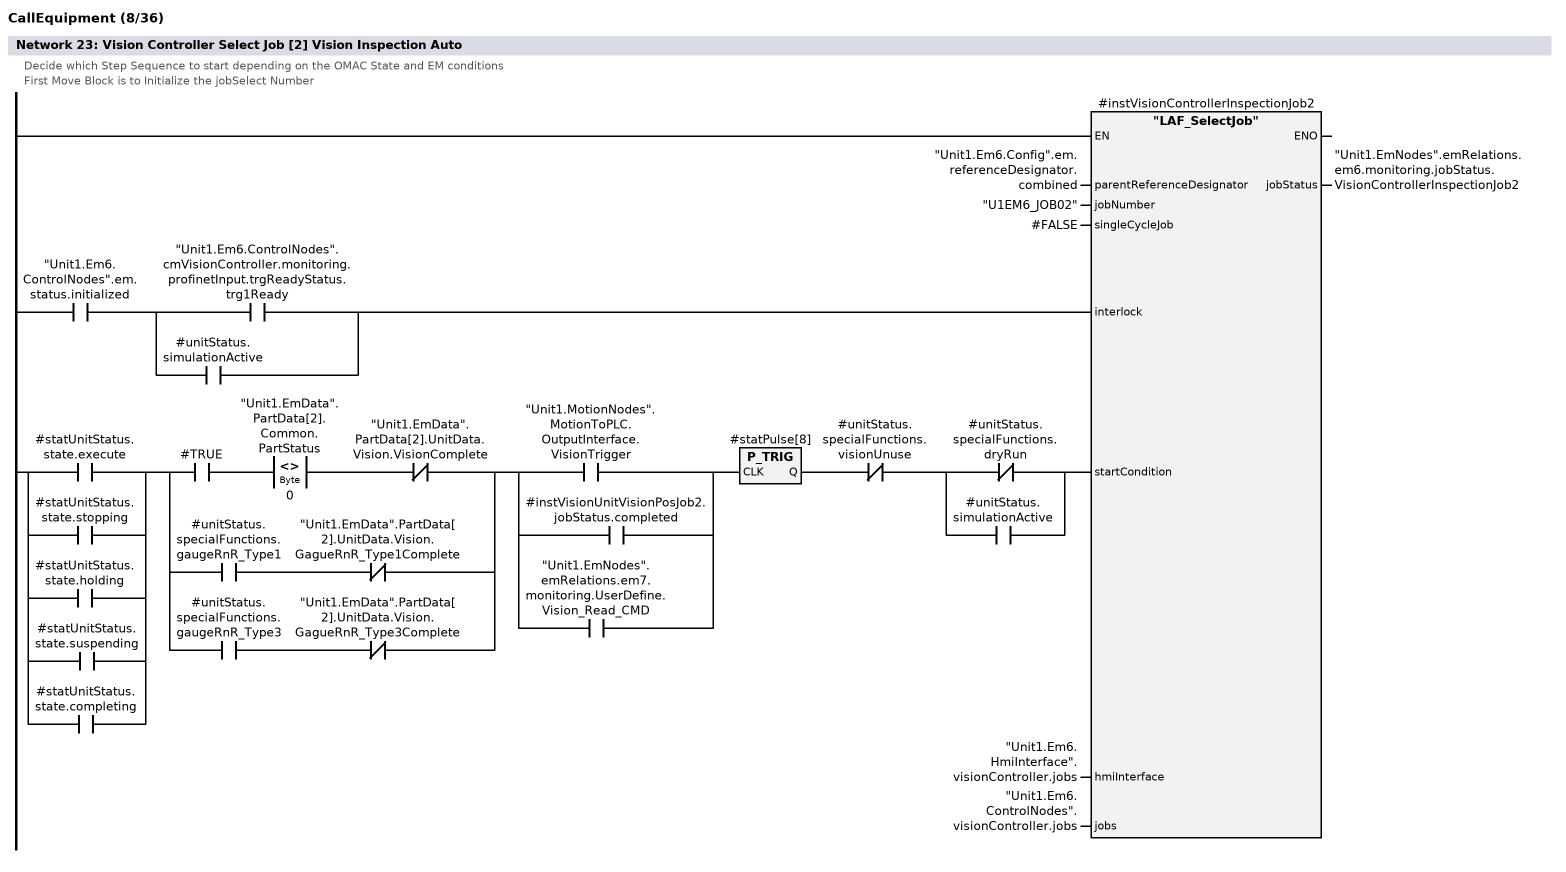
   RUNG wire#powerrail
      #instVisionControllerInspectionJob2(interlock := wire#w2, startCondition := wire#w7, parentReferenceDesignator := "Unit1.Em6.Config".em.referenceDesignator.combined, jobNumber := "U1EM6_JOB02", singleCycleJob := #FALSE, hmiInterface := "Unit1.Em6.HmiInterface".visionController.jobs, jobs := "Unit1.Em6.ControlNodes".visionController.jobs, jobStatus => "Unit1.EmNodes".emRelations.em6.monitoring.jobStatus.VisionControllerInspectionJob2)
   END_RUNG
   RUNG wire#powerrail
      Contact( "Unit1.Em6.ControlNodes".em.status.initialized )
      wire#w1
      Contact( "Unit1.Em6.ControlNodes".cmVisionController.monitoring.profinetInput.trgReadyStatus.trg1Ready )
   END_RUNG wire#w2
   RUNG wire#w1
      Contact( #unitStatus.simulationActive )
   END_RUNG wire#w2
   RUNG wire#powerrail
      Contact( #statUnitStatus.state.execute )
      wire#w3
      Contact( #TRUE )
      { S7_Templates := "SrcType := Byte" } NE_Contact(in1 := "Unit1.EmData".PartData[2].Common.PartStatus, in2 := 0)
      I_Contact( "Unit1.EmData".PartData[2].UnitData.Vision.VisionComplete )
      wire#w4
      Contact( "Unit1.MotionNodes".MotionToPLC.OutputInterface.VisionTrigger )
      wire#w5
      P_Trig( #statPulse[8] )
      I_Contact( #unitStatus.specialFunctions.visionUnuse )
      wire#w6
      I_Contact( #unitStatus.specialFunctions.dryRun )
   END_RUNG wire#w7
   RUNG wire#powerrail
      Contact( #statUnitStatus.state.stopping )
   END_RUNG wire#w3
   RUNG wire#powerrail
      Contact( #statUnitStatus.state.holding )
   END_RUNG wire#w3
   RUNG wire#powerrail
      Contact( #statUnitStatus.state.suspending )
   END_RUNG wire#w3
   RUNG wire#powerrail
      Contact( #statUnitStatus.state.completing )
   END_RUNG wire#w3
   RUNG wire#w3
      Contact( #unitStatus.specialFunctions.gaugeRnR_Type1 )
      I_Contact( "Unit1.EmData".PartData[2].UnitData.Vision.GagueRnR_Type1Complete )
   END_RUNG wire#w4
   RUNG wire#w3
      Contact( #unitStatus.specialFunctions.gaugeRnR_Type3 )
      I_Contact( "Unit1.EmData".PartData[2].UnitData.Vision.GagueRnR_Type3Complete )
   END_RUNG wire#w4
   RUNG wire#w4
      Contact( #instVisionUnitVisionPosJob2.jobStatus.completed )
   END_RUNG wire#w5
   RUNG wire#w4
      Contact( "Unit1.EmNodes".emRelations.em7.monitoring.UserDefine.Vision_Read_CMD )
   END_RUNG wire#w5
   RUNG wire#w6
      Contact( #unitStatus.simulationActive )
   END_RUNG wire#w7
   // the same network as SCL:
   #_w1 := (#statUnitStatus.state.execute OR #statUnitStatus.state.stopping OR #statUnitStatus.state.holding OR #statUnitStatus.state.suspending OR #statUnitStatus.state.completing) AND ((#TRUE AND ("Unit1.EmData".PartData[2].Common.PartStatus <> 0) AND NOT "Unit1.EmData".PartData[2].UnitData.Vision.VisionComplete) OR (#unitStatus.specialFunctions.gaugeRnR_Type1 AND NOT "Unit1.EmData".PartData[2].UnitData.Vision.GagueRnR_Type1Complete) OR (#unitStatus.specialFunctions.gaugeRnR_Type3 AND NOT "Unit1.EmData".PartData[2].UnitData.Vision.GagueRnR_Type3Complete)) AND ("Unit1.MotionNodes".MotionToPLC.OutputInterface.VisionTrigger OR #instVisionUnitVisionPosJob2.jobStatus.completed OR "Unit1.EmNodes".emRelations.em7.monitoring.UserDefine.Vision_Read_CMD);
   #_w2 := #_w1 AND NOT #statPulse[8];   // rising edge
   #statPulse[8] := #_w1;
   #instVisionControllerInspectionJob2(parentReferenceDesignator := "Unit1.Em6.Config".em.referenceDesignator.combined,   // "LAF_SelectJob"
                           jobNumber := "U1EM6_JOB02",
                           singleCycleJob := #FALSE,
                           interlock := "Unit1.Em6.ControlNodes".em.status.initialized AND ("Unit1.Em6.ControlNodes".cmVisionController.monitoring.profinetInput.trgReadyStatus.trg1Ready OR #unitStatus.simulationActive),
                           startCondition := #_w2 AND NOT #unitStatus.specialFunctions.visionUnuse AND (NOT #unitStatus.specialFunctions.dryRun OR #unitStatus.simulationActive),
                           hmiInterface := "Unit1.Em6.HmiInterface".visionController.jobs,
                           jobs := "Unit1.Em6.ControlNodes".visionController.jobs,
                           jobStatus => "Unit1.EmNodes".emRelations.em6.monitoring.jobStatus.VisionControllerInspectionJob2);
END_REGION

REGION Network 24: QrRead Select Job [1] Initialized
   // Decide which Step Sequence to start depending on the OMAC State and EM conditions
   // First Move Block is to Initialize the jobSelect Number
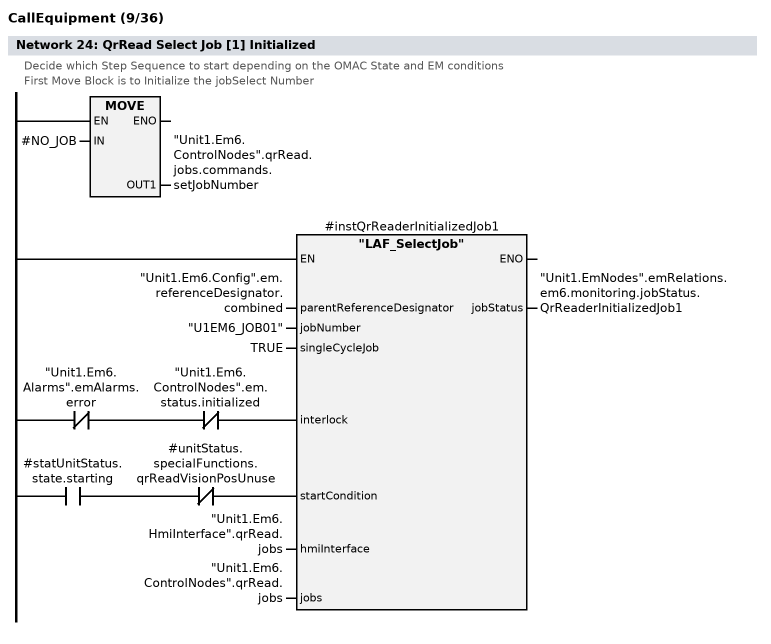
   RUNG wire#powerrail
      Move(in := #NO_JOB, out1 => "Unit1.Em6.ControlNodes".qrRead.jobs.commands.setJobNumber)
   END_RUNG
   RUNG wire#powerrail
      #instQrReaderInitializedJob1(interlock := wire#w1, startCondition := wire#w2, parentReferenceDesignator := "Unit1.Em6.Config".em.referenceDesignator.combined, jobNumber := "U1EM6_JOB01", singleCycleJob := TRUE, hmiInterface := "Unit1.Em6.HmiInterface".qrRead.jobs, jobs := "Unit1.Em6.ControlNodes".qrRead.jobs, jobStatus => "Unit1.EmNodes".emRelations.em6.monitoring.jobStatus.QrReaderInitializedJob1)
   END_RUNG
   RUNG wire#powerrail
      I_Contact( "Unit1.Em6.Alarms".emAlarms.error )
      I_Contact( "Unit1.Em6.ControlNodes".em.status.initialized )
   END_RUNG wire#w1
   RUNG wire#powerrail
      Contact( #statUnitStatus.state.starting )
      I_Contact( #unitStatus.specialFunctions.qrReadVisionPosUnuse )
   END_RUNG wire#w2
   // the same network as SCL:
   "Unit1.Em6.ControlNodes".qrRead.jobs.commands.setJobNumber := #NO_JOB;
   #instQrReaderInitializedJob1(parentReferenceDesignator := "Unit1.Em6.Config".em.referenceDesignator.combined,   // "LAF_SelectJob"
                           jobNumber := "U1EM6_JOB01",
                           singleCycleJob := TRUE,
                           interlock := NOT "Unit1.Em6.Alarms".emAlarms.error AND NOT "Unit1.Em6.ControlNodes".em.status.initialized,
                           startCondition := #statUnitStatus.state.starting AND NOT #unitStatus.specialFunctions.qrReadVisionPosUnuse,
                           hmiInterface := "Unit1.Em6.HmiInterface".qrRead.jobs,
                           jobs := "Unit1.Em6.ControlNodes".qrRead.jobs,
                           jobStatus => "Unit1.EmNodes".emRelations.em6.monitoring.jobStatus.QrReaderInitializedJob1);
END_REGION

REGION Network 25: QrRead Select Job [2] QR Read Auto
   // Decide which Step Sequence to start depending on the OMAC State and EM conditions
   // First Move Block is to Initialize the jobSelect Number
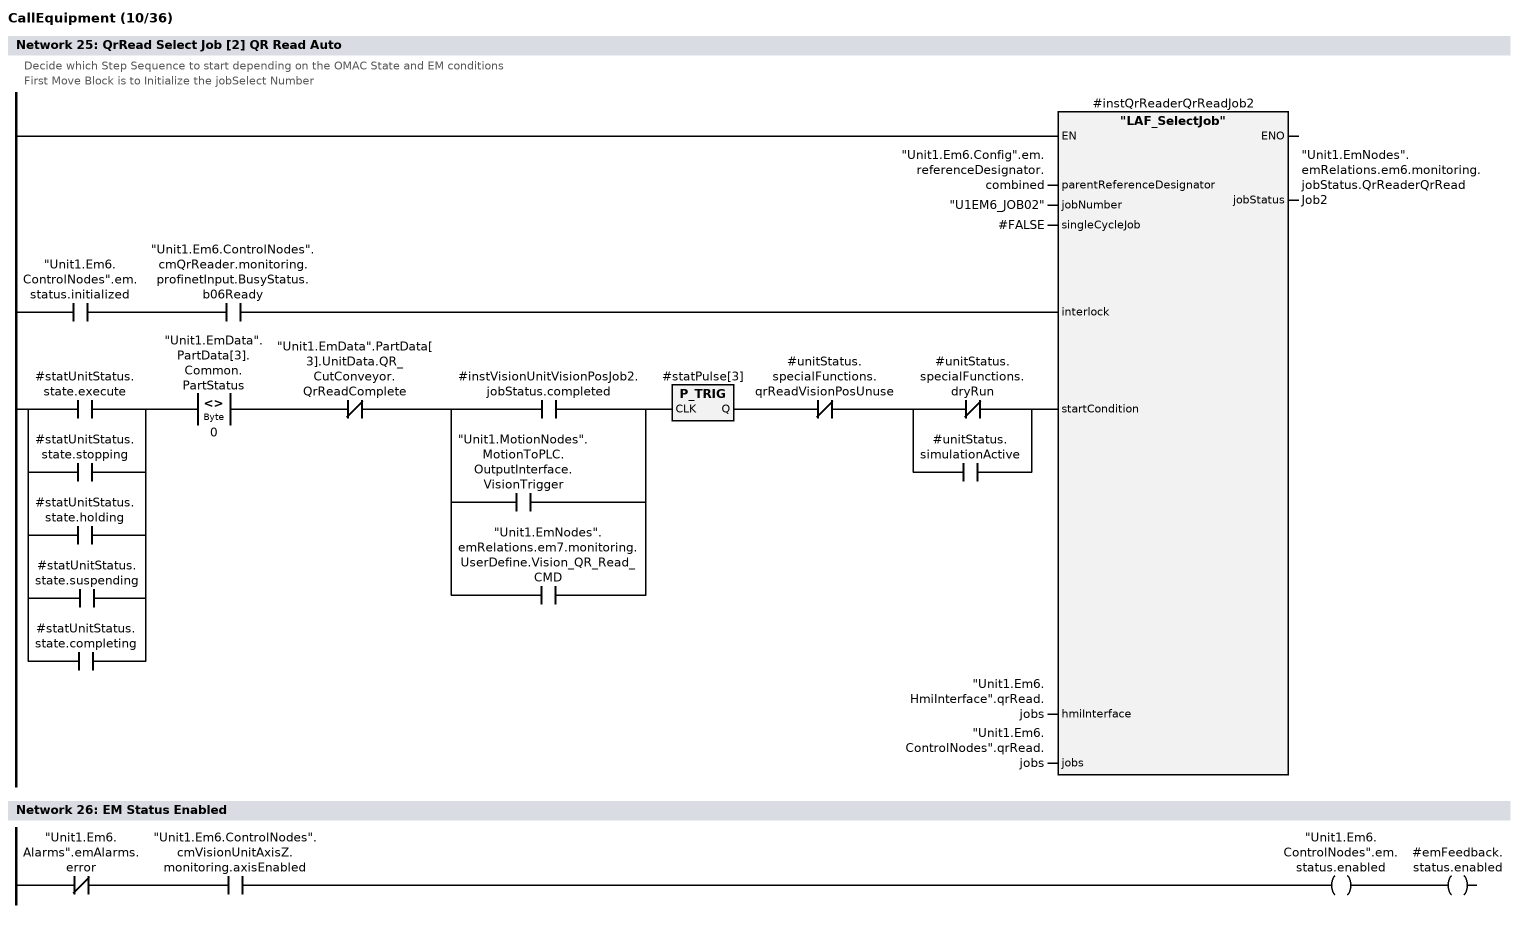
   RUNG wire#powerrail
      #instQrReaderQrReadJob2(interlock := wire#w1, startCondition := wire#w6, parentReferenceDesignator := "Unit1.Em6.Config".em.referenceDesignator.combined, jobNumber := "U1EM6_JOB02", singleCycleJob := #FALSE, hmiInterface := "Unit1.Em6.HmiInterface".qrRead.jobs, jobs := "Unit1.Em6.ControlNodes".qrRead.jobs, jobStatus => "Unit1.EmNodes".emRelations.em6.monitoring.jobStatus.QrReaderQrReadJob2)
   END_RUNG
   RUNG wire#powerrail
      Contact( "Unit1.Em6.ControlNodes".em.status.initialized )
      Contact( "Unit1.Em6.ControlNodes".cmQrReader.monitoring.profinetInput.BusyStatus.b06Ready )
   END_RUNG wire#w1
   RUNG wire#powerrail
      Contact( #statUnitStatus.state.execute )
      wire#w2
      { S7_Templates := "SrcType := Byte" } NE_Contact(in1 := "Unit1.EmData".PartData[3].Common.PartStatus, in2 := 0)
      I_Contact( "Unit1.EmData".PartData[3].UnitData.QR_CutConveyor.QrReadComplete )
      wire#w3
      Contact( #instVisionUnitVisionPosJob2.jobStatus.completed )
      wire#w4
      P_Trig( #statPulse[3] )
      I_Contact( #unitStatus.specialFunctions.qrReadVisionPosUnuse )
      wire#w5
      I_Contact( #unitStatus.specialFunctions.dryRun )
   END_RUNG wire#w6
   RUNG wire#powerrail
      Contact( #statUnitStatus.state.stopping )
   END_RUNG wire#w2
   RUNG wire#powerrail
      Contact( #statUnitStatus.state.holding )
   END_RUNG wire#w2
   RUNG wire#powerrail
      Contact( #statUnitStatus.state.suspending )
   END_RUNG wire#w2
   RUNG wire#powerrail
      Contact( #statUnitStatus.state.completing )
   END_RUNG wire#w2
   RUNG wire#w3
      Contact( "Unit1.MotionNodes".MotionToPLC.OutputInterface.VisionTrigger )
   END_RUNG wire#w4
   RUNG wire#w3
      Contact( "Unit1.EmNodes".emRelations.em7.monitoring.UserDefine.Vision_QR_Read_CMD )
   END_RUNG wire#w4
   RUNG wire#w5
      Contact( #unitStatus.simulationActive )
   END_RUNG wire#w6
   // the same network as SCL:
   #_w1 := (#statUnitStatus.state.execute OR #statUnitStatus.state.stopping OR #statUnitStatus.state.holding OR #statUnitStatus.state.suspending OR #statUnitStatus.state.completing) AND ("Unit1.EmData".PartData[3].Common.PartStatus <> 0) AND NOT "Unit1.EmData".PartData[3].UnitData.QR_CutConveyor.QrReadComplete AND (#instVisionUnitVisionPosJob2.jobStatus.completed OR "Unit1.MotionNodes".MotionToPLC.OutputInterface.VisionTrigger OR "Unit1.EmNodes".emRelations.em7.monitoring.UserDefine.Vision_QR_Read_CMD);
   #_w2 := #_w1 AND NOT #statPulse[3];   // rising edge
   #statPulse[3] := #_w1;
   #instQrReaderQrReadJob2(parentReferenceDesignator := "Unit1.Em6.Config".em.referenceDesignator.combined,   // "LAF_SelectJob"
                           jobNumber := "U1EM6_JOB02",
                           singleCycleJob := #FALSE,
                           interlock := "Unit1.Em6.ControlNodes".em.status.initialized AND "Unit1.Em6.ControlNodes".cmQrReader.monitoring.profinetInput.BusyStatus.b06Ready,
                           startCondition := #_w2 AND NOT #unitStatus.specialFunctions.qrReadVisionPosUnuse AND (NOT #unitStatus.specialFunctions.dryRun OR #unitStatus.simulationActive),
                           hmiInterface := "Unit1.Em6.HmiInterface".qrRead.jobs,
                           jobs := "Unit1.Em6.ControlNodes".qrRead.jobs,
                           jobStatus => "Unit1.EmNodes".emRelations.em6.monitoring.jobStatus.QrReaderQrReadJob2);
END_REGION

REGION Network 26: EM Status Enabled
   RUNG wire#powerrail
      I_Contact( "Unit1.Em6.Alarms".emAlarms.error )
      Contact( "Unit1.Em6.ControlNodes".cmVisionUnitAxisZ.monitoring.axisEnabled )
      Coil( "Unit1.Em6.ControlNodes".em.status.enabled )
      Coil( #emFeedback.status.enabled )
   END_RUNG
   // the same network as SCL:
   "Unit1.Em6.ControlNodes".em.status.enabled := NOT "Unit1.Em6.Alarms".emAlarms.error AND "Unit1.Em6.ControlNodes".cmVisionUnitAxisZ.monitoring.axisEnabled;
   #emFeedback.status.enabled := "Unit1.Em6.ControlNodes".em.status.enabled;
END_REGION

REGION Network 27: EM Status initialized
   // Set em to initialized here. Usually this is done when the initialization job is completed.
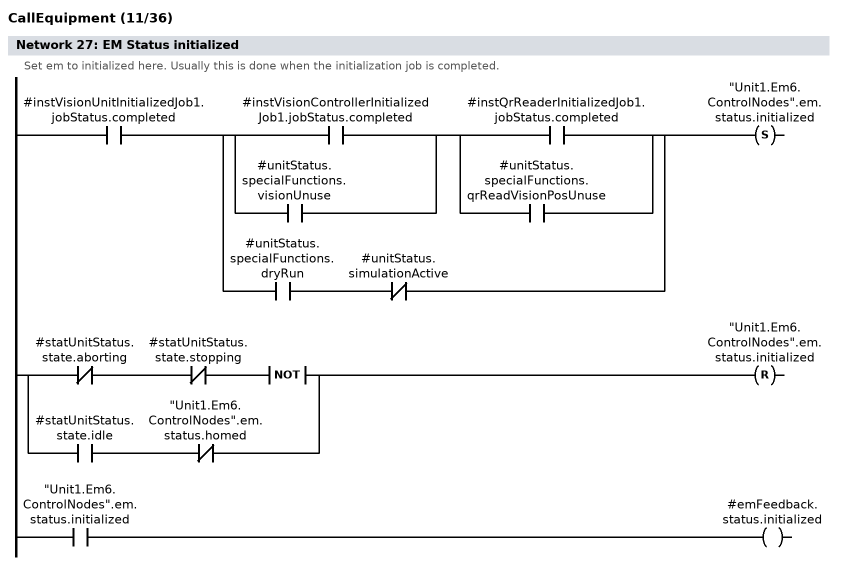
   RUNG wire#powerrail
      Contact( #instVisionUnitInitializedJob1.jobStatus.completed )
      wire#w1
      Contact( #instVisionControllerInitializedJob1.jobStatus.completed )
      wire#w2
      Contact( #instQrReaderInitializedJob1.jobStatus.completed )
      wire#w3
      S_Coil( "Unit1.Em6.ControlNodes".em.status.initialized )
   END_RUNG
   RUNG wire#w1
      Contact( #unitStatus.specialFunctions.visionUnuse )
   END_RUNG wire#w2
   RUNG wire#w2
      Contact( #unitStatus.specialFunctions.qrReadVisionPosUnuse )
   END_RUNG wire#w3
   RUNG wire#w1
      Contact( #unitStatus.specialFunctions.dryRun )
      I_Contact( #unitStatus.simulationActive )
   END_RUNG wire#w3
   RUNG wire#powerrail
      I_Contact( #statUnitStatus.state.aborting )
      I_Contact( #statUnitStatus.state.stopping )
      Not()
      wire#w4
      R_Coil( "Unit1.Em6.ControlNodes".em.status.initialized )
   END_RUNG
   RUNG wire#powerrail
      Contact( #statUnitStatus.state.idle )
      I_Contact( "Unit1.Em6.ControlNodes".em.status.homed )
   END_RUNG wire#w4
   RUNG wire#powerrail
      Contact( "Unit1.Em6.ControlNodes".em.status.initialized )
      Coil( #emFeedback.status.initialized )
   END_RUNG
   // the same network as SCL:
   IF #instVisionUnitInitializedJob1.jobStatus.completed AND (((#instVisionControllerInitializedJob1.jobStatus.completed OR #unitStatus.specialFunctions.visionUnuse) AND (#instQrReaderInitializedJob1.jobStatus.completed OR #unitStatus.specialFunctions.qrReadVisionPosUnuse)) OR (#unitStatus.specialFunctions.dryRun AND NOT #unitStatus.simulationActive)) THEN
       "Unit1.Em6.ControlNodes".em.status.initialized := TRUE;
   END_IF;
   IF NOT (NOT #statUnitStatus.state.aborting AND NOT #statUnitStatus.state.stopping) OR (#statUnitStatus.state.idle AND NOT "Unit1.Em6.ControlNodes".em.status.homed) THEN
       "Unit1.Em6.ControlNodes".em.status.initialized := FALSE;
   END_IF;
   #emFeedback.status.initialized := "Unit1.Em6.ControlNodes".em.status.initialized;
END_REGION

REGION Network 28: EM Status Homed
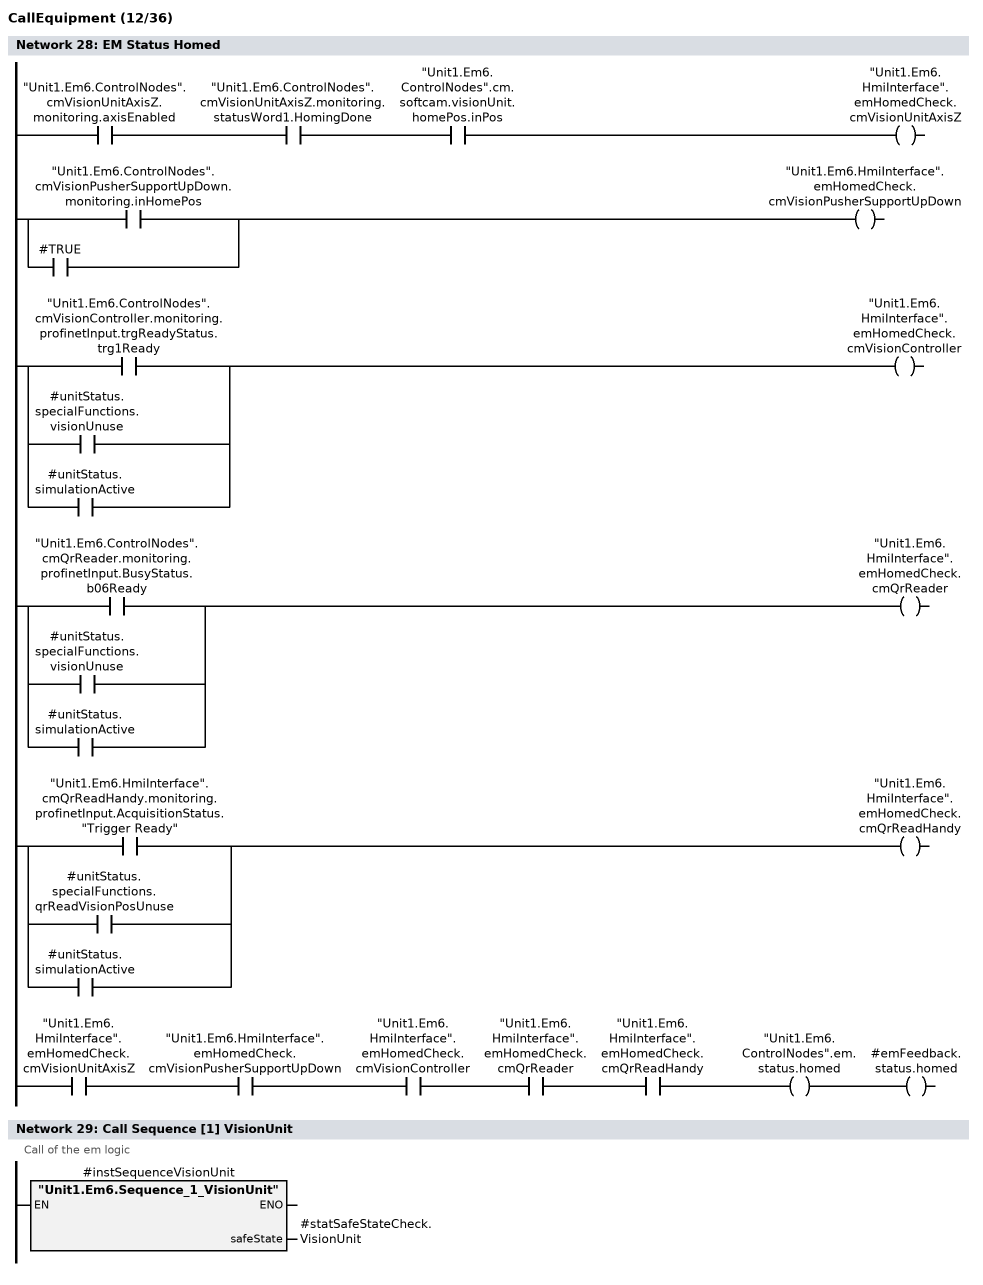
   RUNG wire#powerrail
      Contact( "Unit1.Em6.ControlNodes".cmVisionUnitAxisZ.monitoring.axisEnabled )
      Contact( "Unit1.Em6.ControlNodes".cmVisionUnitAxisZ.monitoring.statusWord1.HomingDone )
      Contact( "Unit1.Em6.ControlNodes".cm.softcam.visionUnit.homePos.inPos )
      Coil( "Unit1.Em6.HmiInterface".emHomedCheck.cmVisionUnitAxisZ )
   END_RUNG
   RUNG wire#powerrail
      Contact( "Unit1.Em6.ControlNodes".cmVisionPusherSupportUpDown.monitoring.inHomePos )
      wire#w1
      Coil( "Unit1.Em6.HmiInterface".emHomedCheck.cmVisionPusherSupportUpDown )
   END_RUNG
   RUNG wire#powerrail
      Contact( #TRUE )
   END_RUNG wire#w1
   RUNG wire#powerrail
      Contact( "Unit1.Em6.ControlNodes".cmVisionController.monitoring.profinetInput.trgReadyStatus.trg1Ready )
      wire#w2
      Coil( "Unit1.Em6.HmiInterface".emHomedCheck.cmVisionController )
   END_RUNG
   RUNG wire#powerrail
      Contact( #unitStatus.specialFunctions.visionUnuse )
   END_RUNG wire#w2
   RUNG wire#powerrail
      Contact( #unitStatus.simulationActive )
   END_RUNG wire#w2
   RUNG wire#powerrail
      Contact( "Unit1.Em6.ControlNodes".cmQrReader.monitoring.profinetInput.BusyStatus.b06Ready )
      wire#w3
      Coil( "Unit1.Em6.HmiInterface".emHomedCheck.cmQrReader )
   END_RUNG
   RUNG wire#powerrail
      Contact( #unitStatus.specialFunctions.visionUnuse )
   END_RUNG wire#w3
   RUNG wire#powerrail
      Contact( #unitStatus.simulationActive )
   END_RUNG wire#w3
   RUNG wire#powerrail
      Contact( "Unit1.Em6.HmiInterface".cmQrReadHandy.monitoring.profinetInput.AcquisitionStatus."Trigger Ready" )
      wire#w4
      Coil( "Unit1.Em6.HmiInterface".emHomedCheck.cmQrReadHandy )
   END_RUNG
   RUNG wire#powerrail
      Contact( #unitStatus.specialFunctions.qrReadVisionPosUnuse )
   END_RUNG wire#w4
   RUNG wire#powerrail
      Contact( #unitStatus.simulationActive )
   END_RUNG wire#w4
   RUNG wire#powerrail
      Contact( "Unit1.Em6.HmiInterface".emHomedCheck.cmVisionUnitAxisZ )
      Contact( "Unit1.Em6.HmiInterface".emHomedCheck.cmVisionPusherSupportUpDown )
      Contact( "Unit1.Em6.HmiInterface".emHomedCheck.cmVisionController )
      Contact( "Unit1.Em6.HmiInterface".emHomedCheck.cmQrReader )
      Contact( "Unit1.Em6.HmiInterface".emHomedCheck.cmQrReadHandy )
      Coil( "Unit1.Em6.ControlNodes".em.status.homed )
      Coil( #emFeedback.status.homed )
   END_RUNG
   // the same network as SCL:
   "Unit1.Em6.HmiInterface".emHomedCheck.cmVisionUnitAxisZ := "Unit1.Em6.ControlNodes".cmVisionUnitAxisZ.monitoring.axisEnabled AND "Unit1.Em6.ControlNodes".cmVisionUnitAxisZ.monitoring.statusWord1.HomingDone AND "Unit1.Em6.ControlNodes".cm.softcam.visionUnit.homePos.inPos;
   "Unit1.Em6.HmiInterface".emHomedCheck.cmVisionPusherSupportUpDown := "Unit1.Em6.ControlNodes".cmVisionPusherSupportUpDown.monitoring.inHomePos OR #TRUE;
   "Unit1.Em6.HmiInterface".emHomedCheck.cmVisionController := "Unit1.Em6.ControlNodes".cmVisionController.monitoring.profinetInput.trgReadyStatus.trg1Ready OR #unitStatus.specialFunctions.visionUnuse OR #unitStatus.simulationActive;
   "Unit1.Em6.HmiInterface".emHomedCheck.cmQrReader := "Unit1.Em6.ControlNodes".cmQrReader.monitoring.profinetInput.BusyStatus.b06Ready OR #unitStatus.specialFunctions.visionUnuse OR #unitStatus.simulationActive;
   "Unit1.Em6.HmiInterface".emHomedCheck.cmQrReadHandy := "Unit1.Em6.HmiInterface".cmQrReadHandy.monitoring.profinetInput.AcquisitionStatus."Trigger Ready" OR #unitStatus.specialFunctions.qrReadVisionPosUnuse OR #unitStatus.simulationActive;
   "Unit1.Em6.ControlNodes".em.status.homed := "Unit1.Em6.HmiInterface".emHomedCheck.cmVisionUnitAxisZ AND "Unit1.Em6.HmiInterface".emHomedCheck.cmVisionPusherSupportUpDown AND "Unit1.Em6.HmiInterface".emHomedCheck.cmVisionController AND "Unit1.Em6.HmiInterface".emHomedCheck.cmQrReader AND "Unit1.Em6.HmiInterface".emHomedCheck.cmQrReadHandy;
   #emFeedback.status.homed := "Unit1.Em6.ControlNodes".em.status.homed;
END_REGION

REGION Network 29: Call Sequence [1] VisionUnit
   // Call of the em logic
   RUNG wire#powerrail
      #instSequenceVisionUnit(safeState => #statSafeStateCheck.VisionUnit)
   END_RUNG
   // the same network as SCL:
   #instSequenceVisionUnit(safeState => #statSafeStateCheck.VisionUnit);   // "Unit1.Em6.Sequence_1_VisionUnit"
END_REGION

REGION Network 30: Call Sequence [2] VisionController
   // Call of the em logic
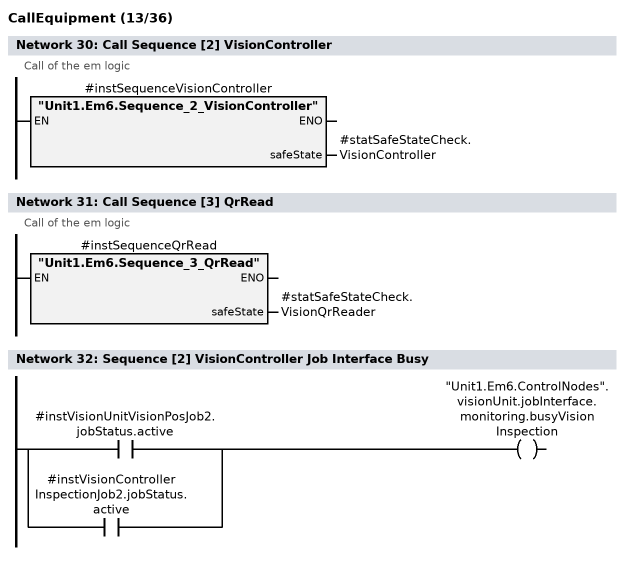
   RUNG wire#powerrail
      #instSequenceVisionController(safeState => #statSafeStateCheck.VisionController)
   END_RUNG
   // the same network as SCL:
   #instSequenceVisionController(safeState => #statSafeStateCheck.VisionController);   // "Unit1.Em6.Sequence_2_VisionController"
END_REGION

REGION Network 31: Call Sequence [3] QrRead
   // Call of the em logic
   RUNG wire#powerrail
      #instSequenceQrRead(safeState => #statSafeStateCheck.VisionQrReader)
   END_RUNG
   // the same network as SCL:
   #instSequenceQrRead(safeState => #statSafeStateCheck.VisionQrReader);   // "Unit1.Em6.Sequence_3_QrRead"
END_REGION

REGION Network 32: Sequence [2] VisionController Job Interface Busy
   RUNG wire#powerrail
      Contact( #instVisionUnitVisionPosJob2.jobStatus.active )
      wire#w1
      Coil( "Unit1.Em6.ControlNodes".visionUnit.jobInterface.monitoring.busyVisionInspection )
   END_RUNG
   RUNG wire#powerrail
      Contact( #instVisionControllerInspectionJob2.jobStatus.active )
   END_RUNG wire#w1
   // the same network as SCL:
   "Unit1.Em6.ControlNodes".visionUnit.jobInterface.monitoring.busyVisionInspection := #instVisionUnitVisionPosJob2.jobStatus.active OR #instVisionControllerInspectionJob2.jobStatus.active;
END_REGION

REGION Network 33: Sequence [2] VisionController Job Interface Done
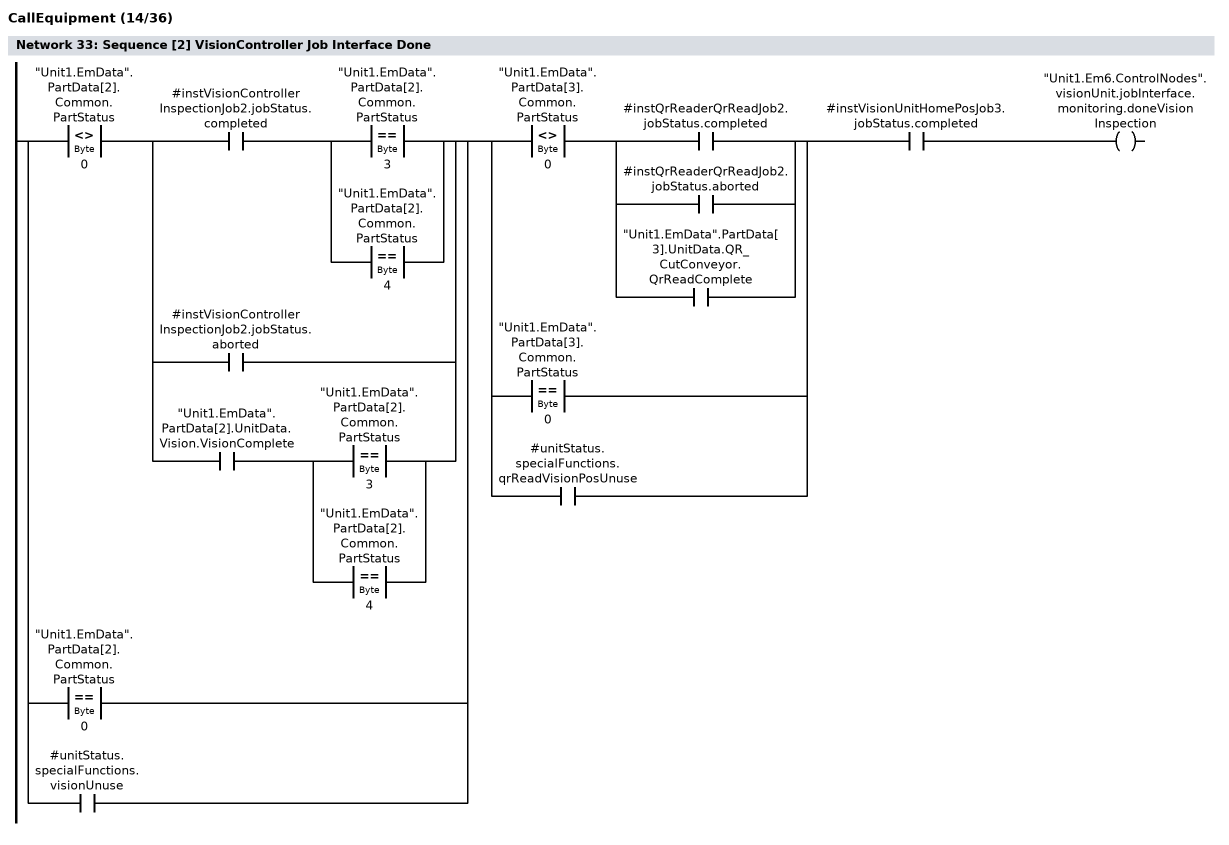
   RUNG wire#powerrail
      { S7_Templates := "SrcType := Byte" } NE_Contact(in1 := "Unit1.EmData".PartData[2].Common.PartStatus, in2 := 0)
      wire#w1
      Contact( #instVisionControllerInspectionJob2.jobStatus.completed )
      wire#w2
      { S7_Templates := "SrcType := Byte" } EQ_Contact(in1 := "Unit1.EmData".PartData[2].Common.PartStatus, in2 := 3)
      wire#w3
      { S7_Templates := "SrcType := Byte" } NE_Contact(in1 := "Unit1.EmData".PartData[3].Common.PartStatus, in2 := 0)
      wire#w5
      Contact( #instQrReaderQrReadJob2.jobStatus.completed )
      wire#w6
      Contact( #instVisionUnitHomePosJob3.jobStatus.completed )
      Coil( "Unit1.Em6.ControlNodes".visionUnit.jobInterface.monitoring.doneVisionInspection )
   END_RUNG
   RUNG wire#w2
      { S7_Templates := "SrcType := Byte" } EQ_Contact(in1 := "Unit1.EmData".PartData[2].Common.PartStatus, in2 := 4)
   END_RUNG wire#w3
   RUNG wire#w1
      Contact( #instVisionControllerInspectionJob2.jobStatus.aborted )
   END_RUNG wire#w3
   RUNG wire#w1
      Contact( "Unit1.EmData".PartData[2].UnitData.Vision.VisionComplete )
      wire#w4
      { S7_Templates := "SrcType := Byte" } EQ_Contact(in1 := "Unit1.EmData".PartData[2].Common.PartStatus, in2 := 3)
   END_RUNG wire#w3
   RUNG wire#w4
      { S7_Templates := "SrcType := Byte" } EQ_Contact(in1 := "Unit1.EmData".PartData[2].Common.PartStatus, in2 := 4)
   END_RUNG wire#w3
   RUNG wire#powerrail
      { S7_Templates := "SrcType := Byte" } EQ_Contact(in1 := "Unit1.EmData".PartData[2].Common.PartStatus, in2 := 0)
   END_RUNG wire#w3
   RUNG wire#powerrail
      Contact( #unitStatus.specialFunctions.visionUnuse )
   END_RUNG wire#w3
   RUNG wire#w5
      Contact( #instQrReaderQrReadJob2.jobStatus.aborted )
   END_RUNG wire#w6
   RUNG wire#w5
      Contact( "Unit1.EmData".PartData[3].UnitData.QR_CutConveyor.QrReadComplete )
   END_RUNG wire#w6
   RUNG wire#w3
      { S7_Templates := "SrcType := Byte" } EQ_Contact(in1 := "Unit1.EmData".PartData[3].Common.PartStatus, in2 := 0)
   END_RUNG wire#w6
   RUNG wire#w3
      Contact( #unitStatus.specialFunctions.qrReadVisionPosUnuse )
   END_RUNG wire#w6
   // the same network as SCL:
   "Unit1.Em6.ControlNodes".visionUnit.jobInterface.monitoring.doneVisionInspection := ((("Unit1.EmData".PartData[2].Common.PartStatus <> 0) AND ((#instVisionControllerInspectionJob2.jobStatus.completed AND (("Unit1.EmData".PartData[2].Common.PartStatus = 3) OR ("Unit1.EmData".PartData[2].Common.PartStatus = 4))) OR #instVisionControllerInspectionJob2.jobStatus.aborted OR ("Unit1.EmData".PartData[2].UnitData.Vision.VisionComplete AND (("Unit1.EmData".PartData[2].Common.PartStatus = 3) OR ("Unit1.EmData".PartData[2].Common.PartStatus = 4))))) OR ("Unit1.EmData".PartData[2].Common.PartStatus = 0) OR #unitStatus.specialFunctions.visionUnuse) AND ((("Unit1.EmData".PartData[3].Common.PartStatus <> 0) AND (#instQrReaderQrReadJob2.jobStatus.completed OR #instQrReaderQrReadJob2.jobStatus.aborted OR "Unit1.EmData".PartData[3].UnitData.QR_CutConveyor.QrReadComplete)) OR ("Unit1.EmData".PartData[3].Common.PartStatus = 0) OR #unitStatus.specialFunctions.qrReadVisionPosUnuse) AND #instVisionUnitHomePosJob3.jobStatus.completed;
END_REGION

REGION Network 34: *************** Axis Velocity Calculate ***************************
END_REGION

REGION Network 35: Call VisionUnit Z Axis
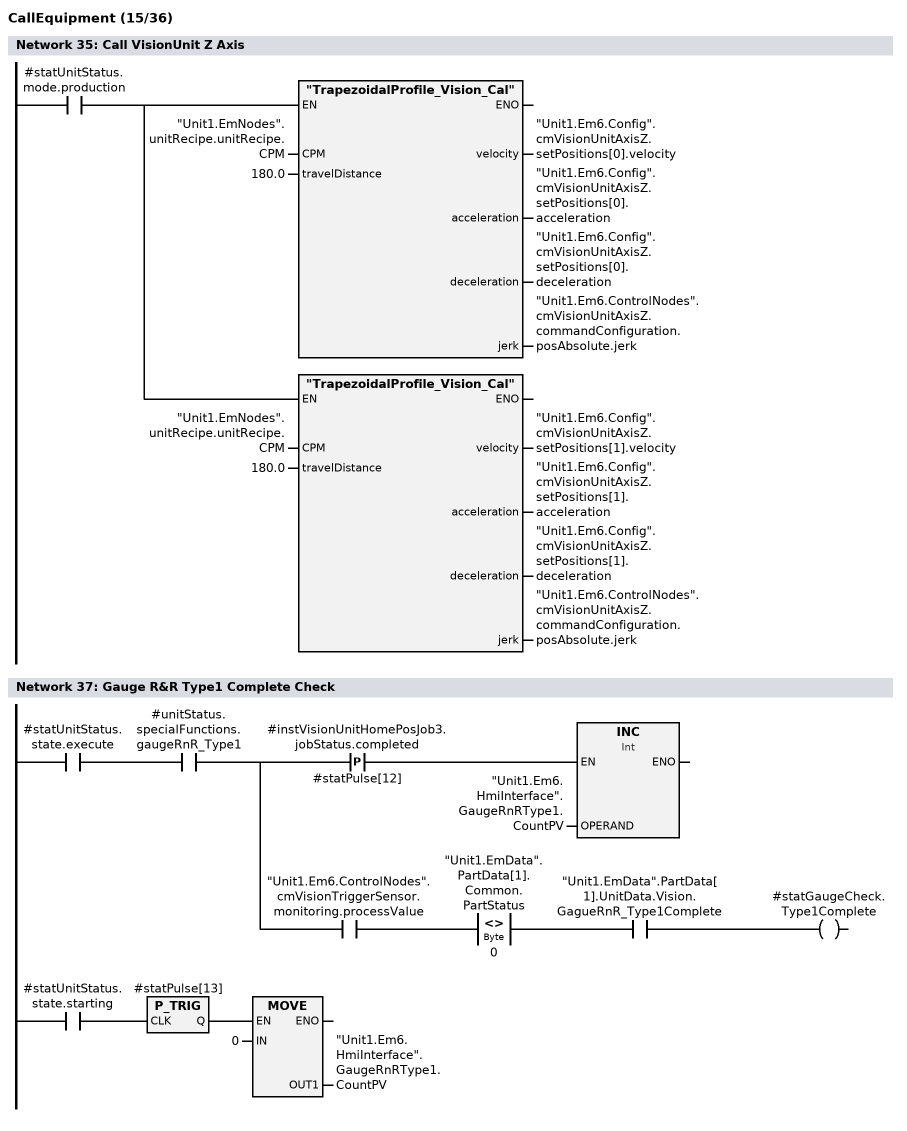
   RUNG wire#powerrail
      Contact( #statUnitStatus.mode.production )
      wire#w1
      "TrapezoidalProfile_Vision_Cal"(CPM := "Unit1.EmNodes".unitRecipe.unitRecipe.CPM, travelDistance := 180.0, velocity => "Unit1.Em6.Config".cmVisionUnitAxisZ.setPositions[0].velocity, acceleration => "Unit1.Em6.Config".cmVisionUnitAxisZ.setPositions[0].acceleration, deceleration => "Unit1.Em6.Config".cmVisionUnitAxisZ.setPositions[0].deceleration, jerk => "Unit1.Em6.ControlNodes".cmVisionUnitAxisZ.commandConfiguration.posAbsolute.jerk)
   END_RUNG
   RUNG wire#w1
      "TrapezoidalProfile_Vision_Cal"(CPM := "Unit1.EmNodes".unitRecipe.unitRecipe.CPM, travelDistance := 180.0, velocity => "Unit1.Em6.Config".cmVisionUnitAxisZ.setPositions[1].velocity, acceleration => "Unit1.Em6.Config".cmVisionUnitAxisZ.setPositions[1].acceleration, deceleration => "Unit1.Em6.Config".cmVisionUnitAxisZ.setPositions[1].deceleration, jerk => "Unit1.Em6.ControlNodes".cmVisionUnitAxisZ.commandConfiguration.posAbsolute.jerk)
   END_RUNG
   // the same network as SCL:
   IF #statUnitStatus.mode.production THEN
       "TrapezoidalProfile_Vision_Cal"(CPM := "Unit1.EmNodes".unitRecipe.unitRecipe.CPM,
                               travelDistance := 180.0,
                               velocity => "Unit1.Em6.Config".cmVisionUnitAxisZ.setPositions[0].velocity,
                               acceleration => "Unit1.Em6.Config".cmVisionUnitAxisZ.setPositions[0].acceleration,
                               deceleration => "Unit1.Em6.Config".cmVisionUnitAxisZ.setPositions[0].deceleration,
                               jerk => "Unit1.Em6.ControlNodes".cmVisionUnitAxisZ.commandConfiguration.posAbsolute.jerk);
       "TrapezoidalProfile_Vision_Cal"(CPM := "Unit1.EmNodes".unitRecipe.unitRecipe.CPM,
                               travelDistance := 180.0,
                               velocity => "Unit1.Em6.Config".cmVisionUnitAxisZ.setPositions[1].velocity,
                               acceleration => "Unit1.Em6.Config".cmVisionUnitAxisZ.setPositions[1].acceleration,
                               deceleration => "Unit1.Em6.Config".cmVisionUnitAxisZ.setPositions[1].deceleration,
                               jerk => "Unit1.Em6.ControlNodes".cmVisionUnitAxisZ.commandConfiguration.posAbsolute.jerk);
   END_IF;
END_REGION

REGION Network 36: ******************** Gague R&R ********************
END_REGION

REGION Network 37: Gauge R&R Type1 Complete Check
   RUNG wire#powerrail
      Contact( #statUnitStatus.state.execute )
      Contact( #unitStatus.specialFunctions.gaugeRnR_Type1 )
      wire#w1
      P_Contact(operand := #instVisionUnitHomePosJob3.jobStatus.completed, bit := #statPulse[12])
      { S7_Templates := "DestType := Int" } Inc( "Unit1.Em6.HmiInterface".GaugeRnRType1.CountPV )
   END_RUNG
   RUNG wire#w1
      Contact( "Unit1.Em6.ControlNodes".cmVisionTriggerSensor.monitoring.processValue )
      { S7_Templates := "SrcType := Byte" } NE_Contact(in1 := "Unit1.EmData".PartData[1].Common.PartStatus, in2 := 0)
      Contact( "Unit1.EmData".PartData[1].UnitData.Vision.GagueRnR_Type1Complete )
      Coil( #statGaugeCheck.Type1Complete )
   END_RUNG
   RUNG wire#powerrail
      Contact( #statUnitStatus.state.starting )
      P_Trig( #statPulse[13] )
      Move(in := 0, out1 => "Unit1.Em6.HmiInterface".GaugeRnRType1.CountPV)
   END_RUNG
   // the same network as SCL:
   #_w1 := #statUnitStatus.state.execute AND #unitStatus.specialFunctions.gaugeRnR_Type1;
   #_w2 := #_w1 AND #instVisionUnitHomePosJob3.jobStatus.completed AND NOT #statPulse[12];   // rising edge of #instVisionUnitHomePosJob3.jobStatus.completed
   #statPulse[12] := #instVisionUnitHomePosJob3.jobStatus.completed;
   IF #_w2 THEN
       "Unit1.Em6.HmiInterface".GaugeRnRType1.CountPV := "Unit1.Em6.HmiInterface".GaugeRnRType1.CountPV + 1;
   END_IF;
   #statGaugeCheck.Type1Complete := #_w1 AND "Unit1.Em6.ControlNodes".cmVisionTriggerSensor.monitoring.processValue AND ("Unit1.EmData".PartData[1].Common.PartStatus <> 0) AND "Unit1.EmData".PartData[1].UnitData.Vision.GagueRnR_Type1Complete;
   #_w3 := #statUnitStatus.state.starting AND NOT #statPulse[13];   // rising edge
   #statPulse[13] := #statUnitStatus.state.starting;
   IF #_w3 THEN "Unit1.Em6.HmiInterface".GaugeRnRType1.CountPV := 0; END_IF;
END_REGION

REGION Network 38: Gauge R&R Type3 Complete Check
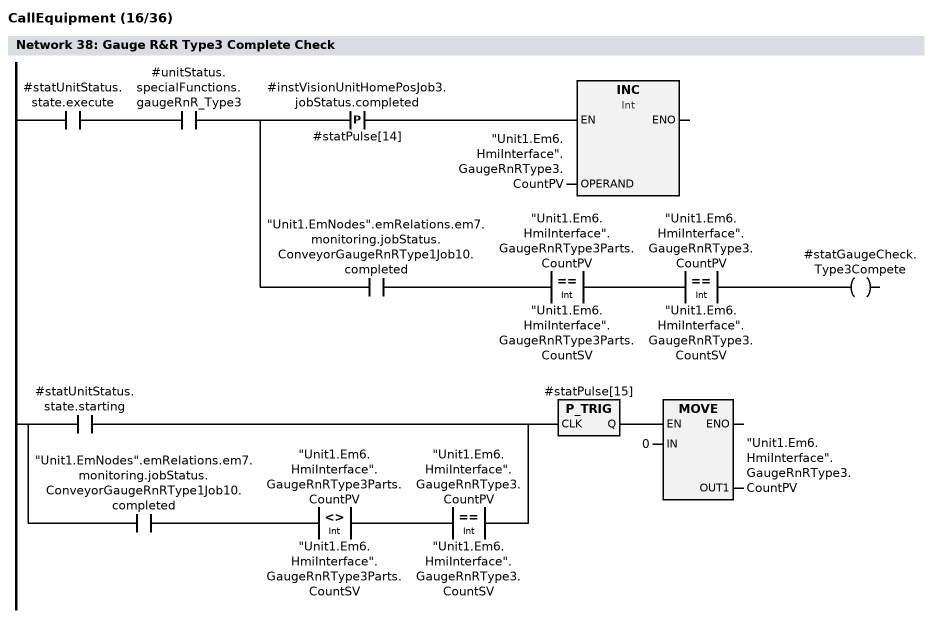
   RUNG wire#powerrail
      Contact( #statUnitStatus.state.execute )
      Contact( #unitStatus.specialFunctions.gaugeRnR_Type3 )
      wire#w1
      P_Contact(operand := #instVisionUnitHomePosJob3.jobStatus.completed, bit := #statPulse[14])
      { S7_Templates := "DestType := Int" } Inc( "Unit1.Em6.HmiInterface".GaugeRnRType3.CountPV )
   END_RUNG
   RUNG wire#w1
      Contact( "Unit1.EmNodes".emRelations.em7.monitoring.jobStatus.ConveyorGaugeRnRType1Job10.completed )
      { S7_Templates := "SrcType := Int" } EQ_Contact(in1 := "Unit1.Em6.HmiInterface".GaugeRnRType3Parts.CountPV, in2 := "Unit1.Em6.HmiInterface".GaugeRnRType3Parts.CountSV)
      { S7_Templates := "SrcType := Int" } EQ_Contact(in1 := "Unit1.Em6.HmiInterface".GaugeRnRType3.CountPV, in2 := "Unit1.Em6.HmiInterface".GaugeRnRType3.CountSV)
      Coil( #statGaugeCheck.Type3Compete )
   END_RUNG
   RUNG wire#powerrail
      Contact( #statUnitStatus.state.starting )
      wire#w2
      P_Trig( #statPulse[15] )
      Move(in := 0, out1 => "Unit1.Em6.HmiInterface".GaugeRnRType3.CountPV)
   END_RUNG
   RUNG wire#powerrail
      Contact( "Unit1.EmNodes".emRelations.em7.monitoring.jobStatus.ConveyorGaugeRnRType1Job10.completed )
      { S7_Templates := "SrcType := Int" } NE_Contact(in1 := "Unit1.Em6.HmiInterface".GaugeRnRType3Parts.CountPV, in2 := "Unit1.Em6.HmiInterface".GaugeRnRType3Parts.CountSV)
      { S7_Templates := "SrcType := Int" } EQ_Contact(in1 := "Unit1.Em6.HmiInterface".GaugeRnRType3.CountPV, in2 := "Unit1.Em6.HmiInterface".GaugeRnRType3.CountSV)
   END_RUNG wire#w2
   // the same network as SCL:
   #_w1 := #statUnitStatus.state.execute AND #unitStatus.specialFunctions.gaugeRnR_Type3;
   #_w2 := #_w1 AND #instVisionUnitHomePosJob3.jobStatus.completed AND NOT #statPulse[14];   // rising edge of #instVisionUnitHomePosJob3.jobStatus.completed
   #statPulse[14] := #instVisionUnitHomePosJob3.jobStatus.completed;
   IF #_w2 THEN
       "Unit1.Em6.HmiInterface".GaugeRnRType3.CountPV := "Unit1.Em6.HmiInterface".GaugeRnRType3.CountPV + 1;
   END_IF;
   #statGaugeCheck.Type3Compete := #_w1 AND "Unit1.EmNodes".emRelations.em7.monitoring.jobStatus.ConveyorGaugeRnRType1Job10.completed AND ("Unit1.Em6.HmiInterface".GaugeRnRType3Parts.CountPV = "Unit1.Em6.HmiInterface".GaugeRnRType3Parts.CountSV) AND ("Unit1.Em6.HmiInterface".GaugeRnRType3.CountPV = "Unit1.Em6.HmiInterface".GaugeRnRType3.CountSV);
   #_w3 := #statUnitStatus.state.starting OR ("Unit1.EmNodes".emRelations.em7.monitoring.jobStatus.ConveyorGaugeRnRType1Job10.completed AND ("Unit1.Em6.HmiInterface".GaugeRnRType3Parts.CountPV <> "Unit1.Em6.HmiInterface".GaugeRnRType3Parts.CountSV) AND ("Unit1.Em6.HmiInterface".GaugeRnRType3.CountPV = "Unit1.Em6.HmiInterface".GaugeRnRType3.CountSV));
   #_w4 := #_w3 AND NOT #statPulse[15];   // rising edge
   #statPulse[15] := #_w3;
   IF #_w4 THEN "Unit1.Em6.HmiInterface".GaugeRnRType3.CountPV := 0; END_IF;
END_REGION

REGION Network 39: ******************** Part Data Generate ********************
END_REGION

REGION Network 40: Call PartData_VisionTriggerPos
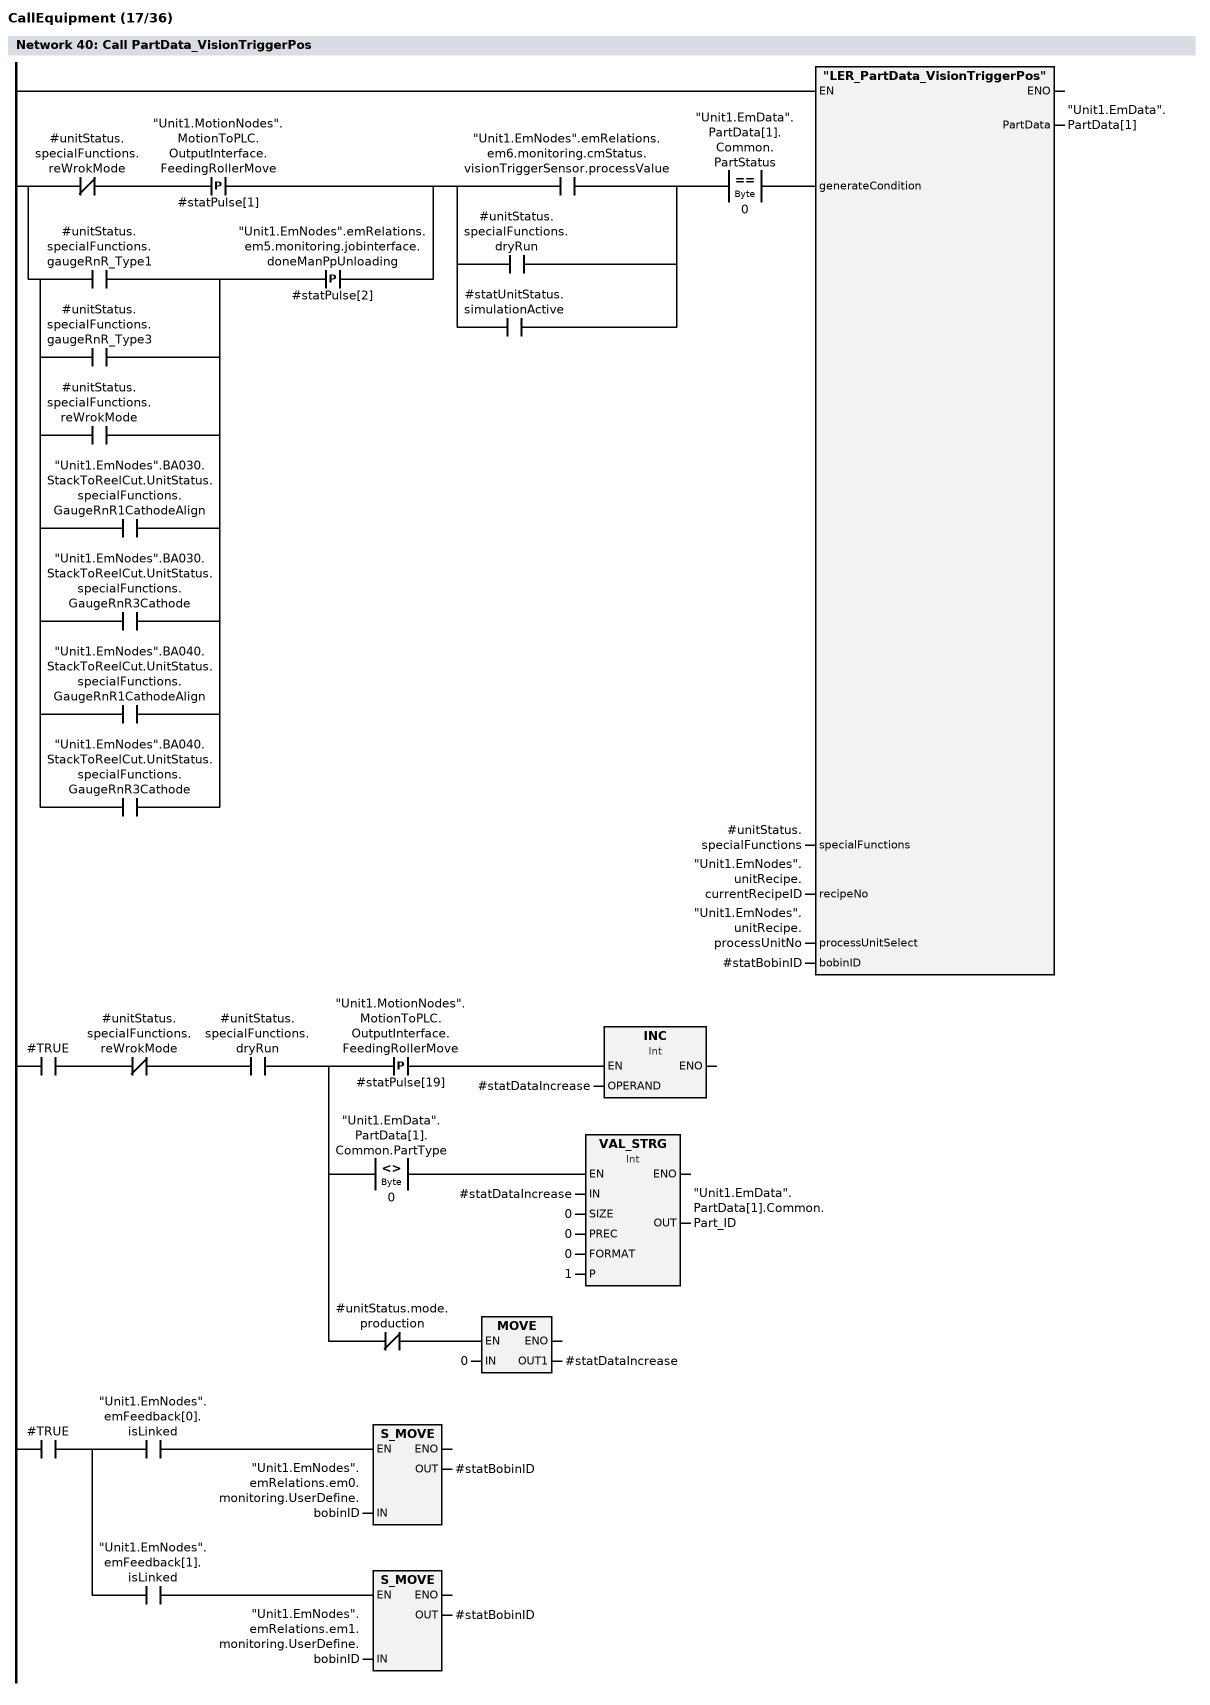
   RUNG wire#powerrail
      "LER_PartData_VisionTriggerPos"(generateCondition := wire#w4, specialFunctions := #unitStatus.specialFunctions, recipeNo := "Unit1.EmNodes".unitRecipe.currentRecipeID, processUnitSelect := "Unit1.EmNodes".unitRecipe.processUnitNo, bobinID := #statBobinID, PartData => "Unit1.EmData".PartData[1])
   END_RUNG
   RUNG wire#powerrail
      I_Contact( #unitStatus.specialFunctions.reWrokMode )
      P_Contact(operand := "Unit1.MotionNodes".MotionToPLC.OutputInterface.FeedingRollerMove, bit := #statPulse[1])
      wire#w1
      Contact( "Unit1.EmNodes".emRelations.em6.monitoring.cmStatus.visionTriggerSensor.processValue )
      wire#w3
      { S7_Templates := "SrcType := Byte" } EQ_Contact(in1 := "Unit1.EmData".PartData[1].Common.PartStatus, in2 := 0)
   END_RUNG wire#w4
   RUNG wire#powerrail
      Contact( #unitStatus.specialFunctions.gaugeRnR_Type1 )
      wire#w2
      P_Contact(operand := "Unit1.EmNodes".emRelations.em5.monitoring.jobinterface.doneManPpUnloading, bit := #statPulse[2])
   END_RUNG wire#w1
   RUNG wire#powerrail
      Contact( #unitStatus.specialFunctions.gaugeRnR_Type3 )
   END_RUNG wire#w2
   RUNG wire#powerrail
      Contact( #unitStatus.specialFunctions.reWrokMode )
   END_RUNG wire#w2
   RUNG wire#powerrail
      Contact( "Unit1.EmNodes".BA030.StackToReelCut.UnitStatus.specialFunctions.GaugeRnR1CathodeAlign )
   END_RUNG wire#w2
   RUNG wire#powerrail
      Contact( "Unit1.EmNodes".BA030.StackToReelCut.UnitStatus.specialFunctions.GaugeRnR3Cathode )
   END_RUNG wire#w2
   RUNG wire#powerrail
      Contact( "Unit1.EmNodes".BA040.StackToReelCut.UnitStatus.specialFunctions.GaugeRnR1CathodeAlign )
   END_RUNG wire#w2
   RUNG wire#powerrail
      Contact( "Unit1.EmNodes".BA040.StackToReelCut.UnitStatus.specialFunctions.GaugeRnR3Cathode )
   END_RUNG wire#w2
   RUNG wire#w1
      Contact( #unitStatus.specialFunctions.dryRun )
   END_RUNG wire#w3
   RUNG wire#w1
      Contact( #statUnitStatus.simulationActive )
   END_RUNG wire#w3
   RUNG wire#powerrail
      Contact( #TRUE )
      I_Contact( #unitStatus.specialFunctions.reWrokMode )
      Contact( #unitStatus.specialFunctions.dryRun )
      wire#w5
      P_Contact(operand := "Unit1.MotionNodes".MotionToPLC.OutputInterface.FeedingRollerMove, bit := #statPulse[19])
      { S7_Templates := "DestType := Int" } Inc( #statDataIncrease )
   END_RUNG
   RUNG wire#w5
      { S7_Templates := "SrcType := Byte" } NE_Contact(in1 := "Unit1.EmData".PartData[1].Common.PartType, in2 := 0)
      { S7_Templates := "[value_type := Int, str_type := String]" } VAL_STRG(IN := #statDataIncrease, SIZE := 0, PREC := 0, FORMAT := 0, P := 1, OUT => "Unit1.EmData".PartData[1].Common.Part_ID)
   END_RUNG
   RUNG wire#w5
      I_Contact( #unitStatus.mode.production )
      Move(in := 0, out1 => #statDataIncrease)
   END_RUNG
   RUNG wire#powerrail
      Contact( #TRUE )
      wire#w6
      Contact( "Unit1.EmNodes".emFeedback[0].isLinked )
      S_Move(in := "Unit1.EmNodes".emRelations.em0.monitoring.UserDefine.bobinID, out => #statBobinID)
   END_RUNG
   RUNG wire#w6
      Contact( "Unit1.EmNodes".emFeedback[1].isLinked )
      S_Move(in := "Unit1.EmNodes".emRelations.em1.monitoring.UserDefine.bobinID, out => #statBobinID)
   END_RUNG
   // the same network as SCL:
   #_w1 := NOT #unitStatus.specialFunctions.reWrokMode AND "Unit1.MotionNodes".MotionToPLC.OutputInterface.FeedingRollerMove AND NOT #statPulse[1];   // rising edge of "Unit1.MotionNodes".MotionToPLC.OutputInterface.FeedingRollerMove
   #statPulse[1] := "Unit1.MotionNodes".MotionToPLC.OutputInterface.FeedingRollerMove;
   #_w2 := (#unitStatus.specialFunctions.gaugeRnR_Type1 OR #unitStatus.specialFunctions.gaugeRnR_Type3 OR #unitStatus.specialFunctions.reWrokMode OR "Unit1.EmNodes".BA030.StackToReelCut.UnitStatus.specialFunctions.GaugeRnR1CathodeAlign OR "Unit1.EmNodes".BA030.StackToReelCut.UnitStatus.specialFunctions.GaugeRnR3Cathode OR "Unit1.EmNodes".BA040.StackToReelCut.UnitStatus.specialFunctions.GaugeRnR1CathodeAlign OR "Unit1.EmNodes".BA040.StackToReelCut.UnitStatus.specialFunctions.GaugeRnR3Cathode) AND "Unit1.EmNodes".emRelations.em5.monitoring.jobinterface.doneManPpUnloading AND NOT #statPulse[2];   // rising edge of "Unit1.EmNodes".emRelations.em5.monitoring.jobinterface.doneManPpUnloading
   #statPulse[2] := "Unit1.EmNodes".emRelations.em5.monitoring.jobinterface.doneManPpUnloading;
   "LER_PartData_VisionTriggerPos"(generateCondition := (#_w1 OR #_w2) AND ("Unit1.EmNodes".emRelations.em6.monitoring.cmStatus.visionTriggerSensor.processValue OR #unitStatus.specialFunctions.dryRun OR #statUnitStatus.simulationActive) AND ("Unit1.EmData".PartData[1].Common.PartStatus = 0),
                           specialFunctions := #unitStatus.specialFunctions,
                           recipeNo := "Unit1.EmNodes".unitRecipe.currentRecipeID,
                           processUnitSelect := "Unit1.EmNodes".unitRecipe.processUnitNo,
                           bobinID := #statBobinID,
                           PartData => "Unit1.EmData".PartData[1]);
   #_w3 := #TRUE AND NOT #unitStatus.specialFunctions.reWrokMode AND #unitStatus.specialFunctions.dryRun;
   #_w4 := #_w3 AND "Unit1.MotionNodes".MotionToPLC.OutputInterface.FeedingRollerMove AND NOT #statPulse[19];   // rising edge of "Unit1.MotionNodes".MotionToPLC.OutputInterface.FeedingRollerMove
   #statPulse[19] := "Unit1.MotionNodes".MotionToPLC.OutputInterface.FeedingRollerMove;
   IF #_w4 THEN #statDataIncrease := #statDataIncrease + 1; END_IF;
   IF #_w3 AND ("Unit1.EmData".PartData[1].Common.PartType <> 0) THEN
       VAL_STRG(IN := #statDataIncrease,
                SIZE := 0,
                PREC := 0,
                FORMAT := 0,
                P := 1,
                OUT => "Unit1.EmData".PartData[1].Common.Part_ID);
   END_IF;
   IF #_w3 AND NOT #unitStatus.mode.production THEN #statDataIncrease := 0; END_IF;
   IF #TRUE AND "Unit1.EmNodes".emFeedback[0].isLinked THEN
       #statBobinID := "Unit1.EmNodes".emRelations.em0.monitoring.UserDefine.bobinID;
   END_IF;
   IF #TRUE AND "Unit1.EmNodes".emFeedback[1].isLinked THEN
       #statBobinID := "Unit1.EmNodes".emRelations.em1.monitoring.UserDefine.bobinID;
   END_IF;
END_REGION

REGION Network 41: Call PartData_VisionPos
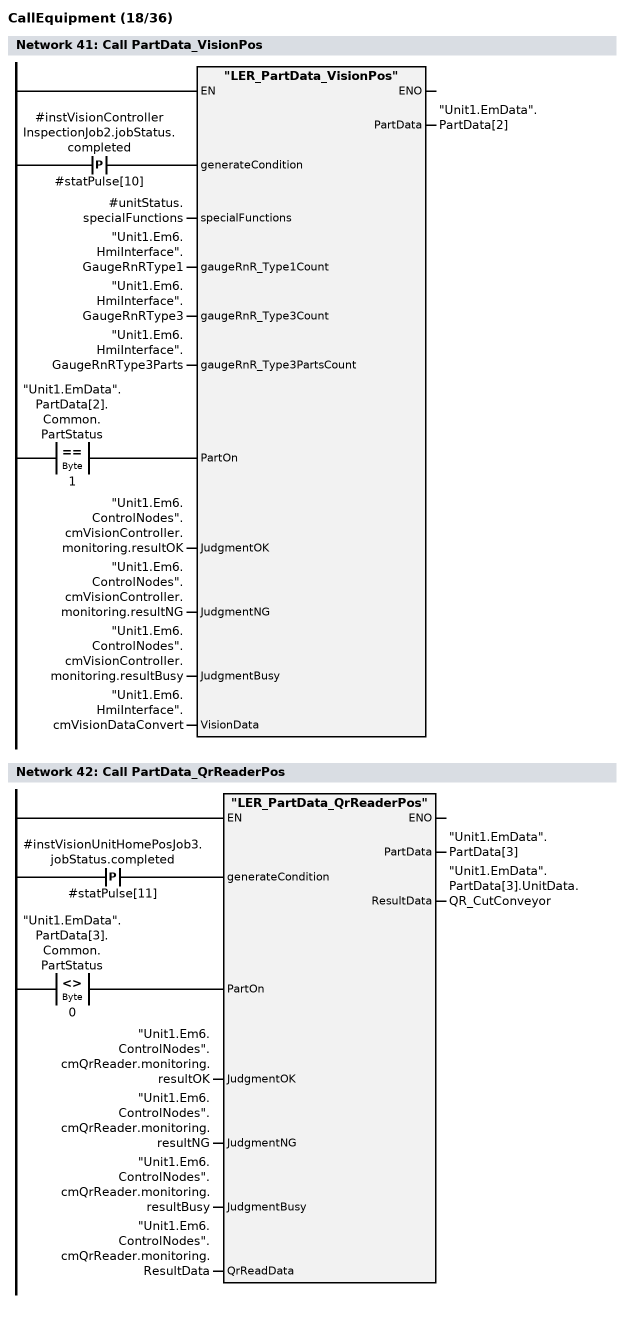
   RUNG wire#powerrail
      "LER_PartData_VisionPos"(generateCondition := wire#w1, PartOn := wire#w2, specialFunctions := #unitStatus.specialFunctions, gaugeRnR_Type1Count := "Unit1.Em6.HmiInterface".GaugeRnRType1, gaugeRnR_Type3Count := "Unit1.Em6.HmiInterface".GaugeRnRType3, gaugeRnR_Type3PartsCount := "Unit1.Em6.HmiInterface".GaugeRnRType3Parts, JudgmentOK := "Unit1.Em6.ControlNodes".cmVisionController.monitoring.resultOK, JudgmentNG := "Unit1.Em6.ControlNodes".cmVisionController.monitoring.resultNG, JudgmentBusy := "Unit1.Em6.ControlNodes".cmVisionController.monitoring.resultBusy, VisionData := "Unit1.Em6.HmiInterface".cmVisionDataConvert, PartData => "Unit1.EmData".PartData[2])
   END_RUNG
   RUNG wire#powerrail
      P_Contact(operand := #instVisionControllerInspectionJob2.jobStatus.completed, bit := #statPulse[10])
   END_RUNG wire#w1
   RUNG wire#powerrail
      { S7_Templates := "SrcType := Byte" } EQ_Contact(in1 := "Unit1.EmData".PartData[2].Common.PartStatus, in2 := 1)
   END_RUNG wire#w2
   // the same network as SCL:
   #_w1 := #instVisionControllerInspectionJob2.jobStatus.completed AND NOT #statPulse[10];   // rising edge of #instVisionControllerInspectionJob2.jobStatus.completed
   #statPulse[10] := #instVisionControllerInspectionJob2.jobStatus.completed;
   "LER_PartData_VisionPos"(generateCondition := #_w1,
                           specialFunctions := #unitStatus.specialFunctions,
                           gaugeRnR_Type1Count := "Unit1.Em6.HmiInterface".GaugeRnRType1,
                           gaugeRnR_Type3Count := "Unit1.Em6.HmiInterface".GaugeRnRType3,
                           gaugeRnR_Type3PartsCount := "Unit1.Em6.HmiInterface".GaugeRnRType3Parts,
                           PartOn := "Unit1.EmData".PartData[2].Common.PartStatus = 1,
                           JudgmentOK := "Unit1.Em6.ControlNodes".cmVisionController.monitoring.resultOK,
                           JudgmentNG := "Unit1.Em6.ControlNodes".cmVisionController.monitoring.resultNG,
                           JudgmentBusy := "Unit1.Em6.ControlNodes".cmVisionController.monitoring.resultBusy,
                           VisionData := "Unit1.Em6.HmiInterface".cmVisionDataConvert,
                           PartData => "Unit1.EmData".PartData[2]);
END_REGION

REGION Network 42: Call PartData_QrReaderPos
   RUNG wire#powerrail
      "LER_PartData_QrReaderPos"(generateCondition := wire#w1, PartOn := wire#w2, JudgmentOK := "Unit1.Em6.ControlNodes".cmQrReader.monitoring.resultOK, JudgmentNG := "Unit1.Em6.ControlNodes".cmQrReader.monitoring.resultNG, JudgmentBusy := "Unit1.Em6.ControlNodes".cmQrReader.monitoring.resultBusy, QrReadData := "Unit1.Em6.ControlNodes".cmQrReader.monitoring.ResultData, PartData => "Unit1.EmData".PartData[3], ResultData => "Unit1.EmData".PartData[3].UnitData.QR_CutConveyor)
   END_RUNG
   RUNG wire#powerrail
      P_Contact(operand := #instVisionUnitHomePosJob3.jobStatus.completed, bit := #statPulse[11])
   END_RUNG wire#w1
   RUNG wire#powerrail
      { S7_Templates := "SrcType := Byte" } NE_Contact(in1 := "Unit1.EmData".PartData[3].Common.PartStatus, in2 := 0)
   END_RUNG wire#w2
   // the same network as SCL:
   #_w1 := #instVisionUnitHomePosJob3.jobStatus.completed AND NOT #statPulse[11];   // rising edge of #instVisionUnitHomePosJob3.jobStatus.completed
   #statPulse[11] := #instVisionUnitHomePosJob3.jobStatus.completed;
   "LER_PartData_QrReaderPos"(generateCondition := #_w1,
                           PartOn := "Unit1.EmData".PartData[3].Common.PartStatus <> 0,
                           JudgmentOK := "Unit1.Em6.ControlNodes".cmQrReader.monitoring.resultOK,
                           JudgmentNG := "Unit1.Em6.ControlNodes".cmQrReader.monitoring.resultNG,
                           JudgmentBusy := "Unit1.Em6.ControlNodes".cmQrReader.monitoring.resultBusy,
                           QrReadData := "Unit1.Em6.ControlNodes".cmQrReader.monitoring.ResultData,
                           PartData => "Unit1.EmData".PartData[3],
                           ResultData => "Unit1.EmData".PartData[3].UnitData.QR_CutConveyor);
END_REGION

REGION Network 43: ******************** Control Modules (Axis) ********************
   // Call control modules that are actuators after the em logic (jobs and sequence), so that the latest commands are applied to the actuators.
END_REGION

REGION Network 44: Reset CMS
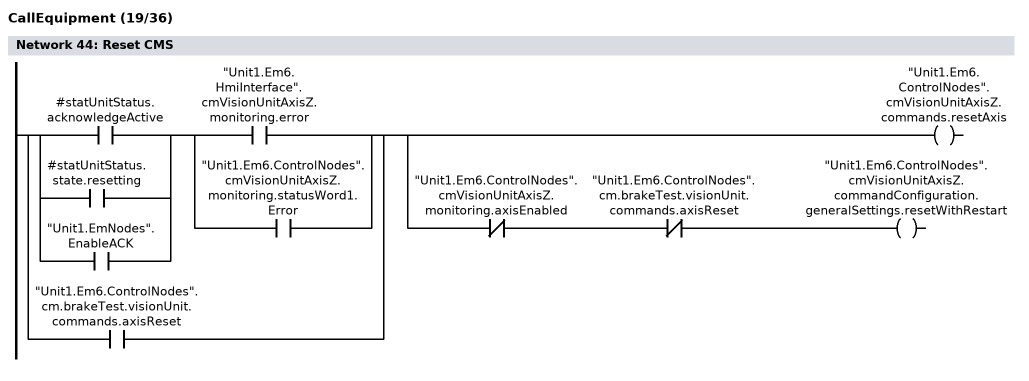
   RUNG wire#powerrail
      Contact( #statUnitStatus.acknowledgeActive )
      wire#w1
      Contact( "Unit1.Em6.HmiInterface".cmVisionUnitAxisZ.monitoring.error )
      wire#w2
      Coil( "Unit1.Em6.ControlNodes".cmVisionUnitAxisZ.commands.resetAxis )
   END_RUNG
   RUNG wire#powerrail
      Contact( #statUnitStatus.state.resetting )
   END_RUNG wire#w1
   RUNG wire#powerrail
      Contact( "Unit1.EmNodes".EnableACK )
   END_RUNG wire#w1
   RUNG wire#w1
      Contact( "Unit1.Em6.ControlNodes".cmVisionUnitAxisZ.monitoring.statusWord1.Error )
   END_RUNG wire#w2
   RUNG wire#powerrail
      Contact( "Unit1.Em6.ControlNodes".cm.brakeTest.visionUnit.commands.axisReset )
   END_RUNG wire#w2
   RUNG wire#w2
      I_Contact( "Unit1.Em6.ControlNodes".cmVisionUnitAxisZ.monitoring.axisEnabled )
      I_Contact( "Unit1.Em6.ControlNodes".cm.brakeTest.visionUnit.commands.axisReset )
      Coil( "Unit1.Em6.ControlNodes".cmVisionUnitAxisZ.commandConfiguration.generalSettings.resetWithRestart )
   END_RUNG
   // the same network as SCL:
   "Unit1.Em6.ControlNodes".cmVisionUnitAxisZ.commands.resetAxis := ((#statUnitStatus.acknowledgeActive OR #statUnitStatus.state.resetting OR "Unit1.EmNodes".EnableACK) AND ("Unit1.Em6.HmiInterface".cmVisionUnitAxisZ.monitoring.error OR "Unit1.Em6.ControlNodes".cmVisionUnitAxisZ.monitoring.statusWord1.Error)) OR "Unit1.Em6.ControlNodes".cm.brakeTest.visionUnit.commands.axisReset;
   "Unit1.Em6.ControlNodes".cmVisionUnitAxisZ.commandConfiguration.generalSettings.resetWithRestart := "Unit1.Em6.ControlNodes".cmVisionUnitAxisZ.commands.resetAxis AND NOT "Unit1.Em6.ControlNodes".cmVisionUnitAxisZ.monitoring.axisEnabled AND NOT "Unit1.Em6.ControlNodes".cm.brakeTest.visionUnit.commands.axisReset;
END_REGION

REGION Network 45: Enable/Disable CMs
   // Enable the axis during the resetting state and disable the axis during the aborting state.
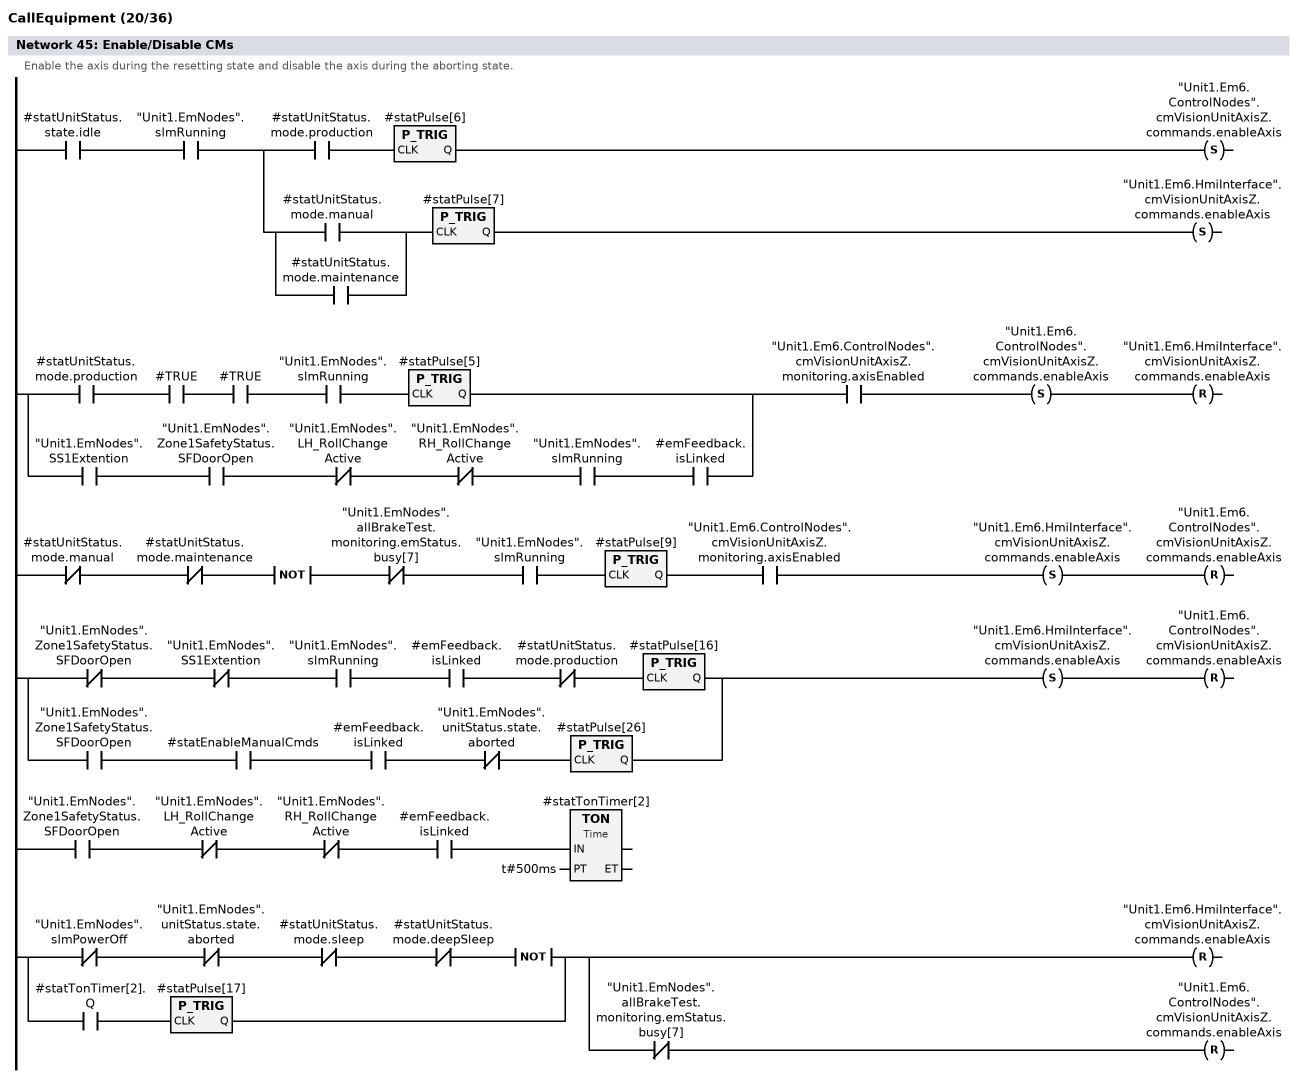
   RUNG wire#powerrail
      Contact( #statUnitStatus.state.idle )
      Contact( "Unit1.EmNodes".slmRunning )
      wire#w1
      Contact( #statUnitStatus.mode.production )
      P_Trig( #statPulse[6] )
      S_Coil( "Unit1.Em6.ControlNodes".cmVisionUnitAxisZ.commands.enableAxis )
   END_RUNG
   RUNG wire#w1
      Contact( #statUnitStatus.mode.manual )
      wire#w2
      P_Trig( #statPulse[7] )
      S_Coil( "Unit1.Em6.HmiInterface".cmVisionUnitAxisZ.commands.enableAxis )
   END_RUNG
   RUNG wire#w1
      Contact( #statUnitStatus.mode.maintenance )
   END_RUNG wire#w2
   RUNG wire#powerrail
      Contact( #statUnitStatus.mode.production )
      Contact( #TRUE )
      Contact( #TRUE )
      Contact( "Unit1.EmNodes".slmRunning )
      P_Trig( #statPulse[5] )
      wire#w3
      Contact( "Unit1.Em6.ControlNodes".cmVisionUnitAxisZ.monitoring.axisEnabled )
      S_Coil( "Unit1.Em6.ControlNodes".cmVisionUnitAxisZ.commands.enableAxis )
      R_Coil( "Unit1.Em6.HmiInterface".cmVisionUnitAxisZ.commands.enableAxis )
   END_RUNG
   RUNG wire#powerrail
      Contact( "Unit1.EmNodes".SS1Extention )
      Contact( "Unit1.EmNodes".Zone1SafetyStatus.SFDoorOpen )
      I_Contact( "Unit1.EmNodes".LH_RollChangeActive )
      I_Contact( "Unit1.EmNodes".RH_RollChangeActive )
      Contact( "Unit1.EmNodes".slmRunning )
      Contact( #emFeedback.isLinked )
   END_RUNG wire#w3
   RUNG wire#powerrail
      I_Contact( #statUnitStatus.mode.manual )
      I_Contact( #statUnitStatus.mode.maintenance )
      Not()
      I_Contact( "Unit1.EmNodes".allBrakeTest.monitoring.emStatus.busy[7] )
      Contact( "Unit1.EmNodes".slmRunning )
      P_Trig( #statPulse[9] )
      Contact( "Unit1.Em6.ControlNodes".cmVisionUnitAxisZ.monitoring.axisEnabled )
      S_Coil( "Unit1.Em6.HmiInterface".cmVisionUnitAxisZ.commands.enableAxis )
      R_Coil( "Unit1.Em6.ControlNodes".cmVisionUnitAxisZ.commands.enableAxis )
   END_RUNG
   RUNG wire#powerrail
      I_Contact( "Unit1.EmNodes".Zone1SafetyStatus.SFDoorOpen )
      I_Contact( "Unit1.EmNodes".SS1Extention )
      Contact( "Unit1.EmNodes".slmRunning )
      Contact( #emFeedback.isLinked )
      I_Contact( #statUnitStatus.mode.production )
      P_Trig( #statPulse[16] )
      wire#w4
      S_Coil( "Unit1.Em6.HmiInterface".cmVisionUnitAxisZ.commands.enableAxis )
      R_Coil( "Unit1.Em6.ControlNodes".cmVisionUnitAxisZ.commands.enableAxis )
   END_RUNG
   RUNG wire#powerrail
      Contact( "Unit1.EmNodes".Zone1SafetyStatus.SFDoorOpen )
      Contact( #statEnableManualCmds )
      Contact( #emFeedback.isLinked )
      I_Contact( "Unit1.EmNodes".unitStatus.state.aborted )
      P_Trig( #statPulse[26] )
   END_RUNG wire#w4
   RUNG wire#powerrail
      Contact( "Unit1.EmNodes".Zone1SafetyStatus.SFDoorOpen )
      I_Contact( "Unit1.EmNodes".LH_RollChangeActive )
      I_Contact( "Unit1.EmNodes".RH_RollChangeActive )
      Contact( #emFeedback.isLinked )
      { S7_Templates := "time_type := Time" } #statTonTimer[2].TON(pt := t#500ms, et =>)
   END_RUNG
   RUNG wire#powerrail
      I_Contact( "Unit1.EmNodes".slmPowerOff )
      I_Contact( "Unit1.EmNodes".unitStatus.state.aborted )
      I_Contact( #statUnitStatus.mode.sleep )
      I_Contact( #statUnitStatus.mode.deepSleep )
      Not()
      wire#w5
      R_Coil( "Unit1.Em6.HmiInterface".cmVisionUnitAxisZ.commands.enableAxis )
   END_RUNG
   RUNG wire#powerrail
      Contact( #statTonTimer[2].Q )
      P_Trig( #statPulse[17] )
   END_RUNG wire#w5
   RUNG wire#w5
      I_Contact( "Unit1.EmNodes".allBrakeTest.monitoring.emStatus.busy[7] )
      R_Coil( "Unit1.Em6.ControlNodes".cmVisionUnitAxisZ.commands.enableAxis )
   END_RUNG
   // the same network as SCL:
   #_w1 := #statUnitStatus.state.idle AND "Unit1.EmNodes".slmRunning;
   #_w2 := #_w1 AND #statUnitStatus.mode.production;
   #_w3 := #_w2 AND NOT #statPulse[6];   // rising edge
   #statPulse[6] := #_w2;
   IF #_w3 THEN "Unit1.Em6.ControlNodes".cmVisionUnitAxisZ.commands.enableAxis := TRUE; END_IF;
   #_w4 := #_w1 AND (#statUnitStatus.mode.manual OR #statUnitStatus.mode.maintenance);
   #_w5 := #_w4 AND NOT #statPulse[7];   // rising edge
   #statPulse[7] := #_w4;
   IF #_w5 THEN "Unit1.Em6.HmiInterface".cmVisionUnitAxisZ.commands.enableAxis := TRUE; END_IF;
   #_w6 := #statUnitStatus.mode.production AND #TRUE AND #TRUE AND "Unit1.EmNodes".slmRunning;
   #_w7 := #_w6 AND NOT #statPulse[5];   // rising edge
   #statPulse[5] := #_w6;
   IF (#_w7 OR ("Unit1.EmNodes".SS1Extention AND "Unit1.EmNodes".Zone1SafetyStatus.SFDoorOpen AND NOT "Unit1.EmNodes".LH_RollChangeActive AND NOT "Unit1.EmNodes".RH_RollChangeActive AND "Unit1.EmNodes".slmRunning AND #emFeedback.isLinked)) AND "Unit1.Em6.ControlNodes".cmVisionUnitAxisZ.monitoring.axisEnabled THEN
       "Unit1.Em6.ControlNodes".cmVisionUnitAxisZ.commands.enableAxis := TRUE;
       "Unit1.Em6.HmiInterface".cmVisionUnitAxisZ.commands.enableAxis := FALSE;
   END_IF;
   #_w8 := NOT (NOT #statUnitStatus.mode.manual AND NOT #statUnitStatus.mode.maintenance) AND NOT "Unit1.EmNodes".allBrakeTest.monitoring.emStatus.busy[7] AND "Unit1.EmNodes".slmRunning;
   #_w9 := #_w8 AND NOT #statPulse[9];   // rising edge
   #statPulse[9] := #_w8;
   IF #_w9 AND "Unit1.Em6.ControlNodes".cmVisionUnitAxisZ.monitoring.axisEnabled THEN
       "Unit1.Em6.HmiInterface".cmVisionUnitAxisZ.commands.enableAxis := TRUE;
       "Unit1.Em6.ControlNodes".cmVisionUnitAxisZ.commands.enableAxis := FALSE;
   END_IF;
   #_w10 := NOT "Unit1.EmNodes".Zone1SafetyStatus.SFDoorOpen AND NOT "Unit1.EmNodes".SS1Extention AND "Unit1.EmNodes".slmRunning AND #emFeedback.isLinked AND NOT #statUnitStatus.mode.production;
   #_w11 := #_w10 AND NOT #statPulse[16];   // rising edge
   #statPulse[16] := #_w10;
   #_w12 := "Unit1.EmNodes".Zone1SafetyStatus.SFDoorOpen AND #statEnableManualCmds AND #emFeedback.isLinked AND NOT "Unit1.EmNodes".unitStatus.state.aborted;
   #_w13 := #_w12 AND NOT #statPulse[26];   // rising edge
   #statPulse[26] := #_w12;
   IF #_w11 OR #_w13 THEN
       "Unit1.Em6.HmiInterface".cmVisionUnitAxisZ.commands.enableAxis := TRUE;
       "Unit1.Em6.ControlNodes".cmVisionUnitAxisZ.commands.enableAxis := FALSE;
   END_IF;
   #statTonTimer[2].TON(IN := "Unit1.EmNodes".Zone1SafetyStatus.SFDoorOpen AND NOT "Unit1.EmNodes".LH_RollChangeActive AND NOT "Unit1.EmNodes".RH_RollChangeActive AND #emFeedback.isLinked,
                        PT := t#500ms);
   #_w14 := #statTonTimer[2].Q AND NOT #statPulse[17];   // rising edge
   #statPulse[17] := #statTonTimer[2].Q;
   #_w15 := NOT (NOT "Unit1.EmNodes".slmPowerOff AND NOT "Unit1.EmNodes".unitStatus.state.aborted AND NOT #statUnitStatus.mode.sleep AND NOT #statUnitStatus.mode.deepSleep) OR #_w14;
   IF #_w15 THEN "Unit1.Em6.HmiInterface".cmVisionUnitAxisZ.commands.enableAxis := FALSE; END_IF;
   IF #_w15 AND NOT "Unit1.EmNodes".allBrakeTest.monitoring.emStatus.busy[7] THEN
       "Unit1.Em6.ControlNodes".cmVisionUnitAxisZ.commands.enableAxis := FALSE;
   END_IF;
END_REGION

REGION Network 46: LBC_Axis64Pos Operation Mode
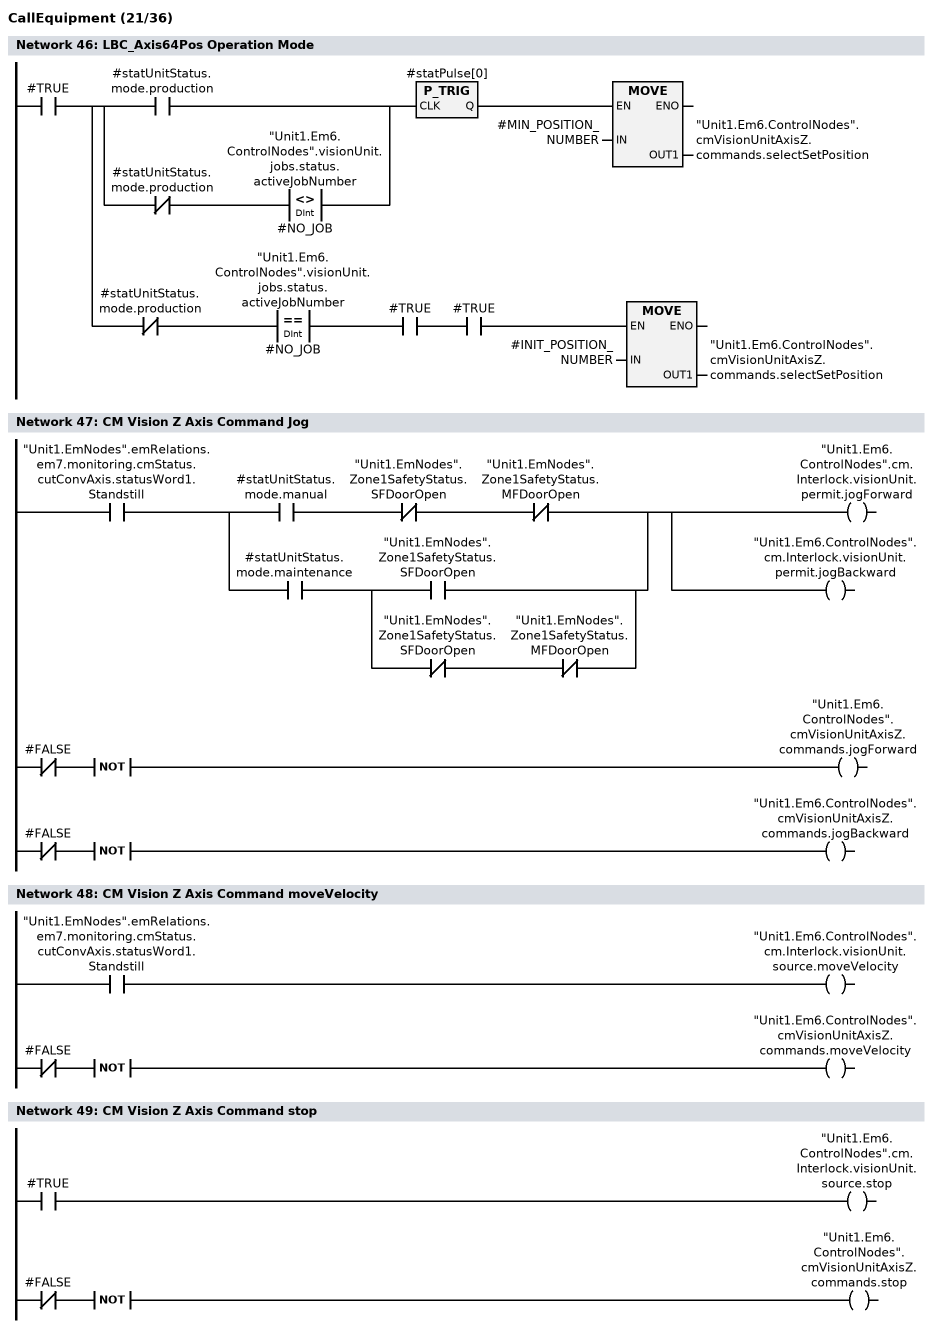
   RUNG wire#powerrail
      Contact( #TRUE )
      wire#w1
      Contact( #statUnitStatus.mode.production )
      wire#w2
      P_Trig( #statPulse[0] )
      Move(in := #MIN_POSITION_NUMBER, out1 => "Unit1.Em6.ControlNodes".cmVisionUnitAxisZ.commands.selectSetPosition)
   END_RUNG
   RUNG wire#w1
      I_Contact( #statUnitStatus.mode.production )
      { S7_Templates := "SrcType := DInt" } NE_Contact(in1 := "Unit1.Em6.ControlNodes".visionUnit.jobs.status.activeJobNumber, in2 := #NO_JOB)
   END_RUNG wire#w2
   RUNG wire#w1
      I_Contact( #statUnitStatus.mode.production )
      { S7_Templates := "SrcType := DInt" } EQ_Contact(in1 := "Unit1.Em6.ControlNodes".visionUnit.jobs.status.activeJobNumber, in2 := #NO_JOB)
      Contact( #TRUE )
      Contact( #TRUE )
      Move(in := #INIT_POSITION_NUMBER, out1 => "Unit1.Em6.ControlNodes".cmVisionUnitAxisZ.commands.selectSetPosition)
   END_RUNG
   // the same network as SCL:
   #_w1 := #TRUE AND (#statUnitStatus.mode.production OR (NOT #statUnitStatus.mode.production AND ("Unit1.Em6.ControlNodes".visionUnit.jobs.status.activeJobNumber <> #NO_JOB)));
   #_w2 := #_w1 AND NOT #statPulse[0];   // rising edge
   #statPulse[0] := #_w1;
   IF #_w2 THEN
       "Unit1.Em6.ControlNodes".cmVisionUnitAxisZ.commands.selectSetPosition := #MIN_POSITION_NUMBER;
   END_IF;
   IF #TRUE AND NOT #statUnitStatus.mode.production AND ("Unit1.Em6.ControlNodes".visionUnit.jobs.status.activeJobNumber = #NO_JOB) AND #TRUE AND #TRUE THEN
       "Unit1.Em6.ControlNodes".cmVisionUnitAxisZ.commands.selectSetPosition := #INIT_POSITION_NUMBER;
   END_IF;
END_REGION

REGION Network 47: CM Vision Z Axis Command Jog
   RUNG wire#powerrail
      Contact( "Unit1.EmNodes".emRelations.em7.monitoring.cmStatus.cutConvAxis.statusWord1.Standstill )
      wire#w1
      Contact( #statUnitStatus.mode.manual )
      I_Contact( "Unit1.EmNodes".Zone1SafetyStatus.SFDoorOpen )
      I_Contact( "Unit1.EmNodes".Zone1SafetyStatus.MFDoorOpen )
      wire#w2
      Coil( "Unit1.Em6.ControlNodes".cm.Interlock.visionUnit.permit.jogForward )
   END_RUNG
   RUNG wire#w1
      Contact( #statUnitStatus.mode.maintenance )
      wire#w3
      Contact( "Unit1.EmNodes".Zone1SafetyStatus.SFDoorOpen )
   END_RUNG wire#w2
   RUNG wire#w3
      I_Contact( "Unit1.EmNodes".Zone1SafetyStatus.SFDoorOpen )
      I_Contact( "Unit1.EmNodes".Zone1SafetyStatus.MFDoorOpen )
   END_RUNG wire#w2
   RUNG wire#w2
      Coil( "Unit1.Em6.ControlNodes".cm.Interlock.visionUnit.permit.jogBackward )
   END_RUNG
   RUNG wire#powerrail
      I_Contact( #FALSE )
      Not()
      Coil( "Unit1.Em6.ControlNodes".cmVisionUnitAxisZ.commands.jogForward )
   END_RUNG
   RUNG wire#powerrail
      I_Contact( #FALSE )
      Not()
      Coil( "Unit1.Em6.ControlNodes".cmVisionUnitAxisZ.commands.jogBackward )
   END_RUNG
   // the same network as SCL:
   "Unit1.Em6.ControlNodes".cm.Interlock.visionUnit.permit.jogForward := "Unit1.EmNodes".emRelations.em7.monitoring.cmStatus.cutConvAxis.statusWord1.Standstill AND ((#statUnitStatus.mode.manual AND NOT "Unit1.EmNodes".Zone1SafetyStatus.SFDoorOpen AND NOT "Unit1.EmNodes".Zone1SafetyStatus.MFDoorOpen) OR (#statUnitStatus.mode.maintenance AND ("Unit1.EmNodes".Zone1SafetyStatus.SFDoorOpen OR (NOT "Unit1.EmNodes".Zone1SafetyStatus.SFDoorOpen AND NOT "Unit1.EmNodes".Zone1SafetyStatus.MFDoorOpen))));
   "Unit1.Em6.ControlNodes".cm.Interlock.visionUnit.permit.jogBackward := "Unit1.Em6.ControlNodes".cm.Interlock.visionUnit.permit.jogForward;
   "Unit1.Em6.ControlNodes".cmVisionUnitAxisZ.commands.jogForward := NOT (NOT #FALSE);
   "Unit1.Em6.ControlNodes".cmVisionUnitAxisZ.commands.jogBackward := NOT (NOT #FALSE);
END_REGION

REGION Network 48: CM Vision Z Axis Command moveVelocity
   RUNG wire#powerrail
      Contact( "Unit1.EmNodes".emRelations.em7.monitoring.cmStatus.cutConvAxis.statusWord1.Standstill )
      Coil( "Unit1.Em6.ControlNodes".cm.Interlock.visionUnit.source.moveVelocity )
   END_RUNG
   RUNG wire#powerrail
      I_Contact( #FALSE )
      Not()
      Coil( "Unit1.Em6.ControlNodes".cmVisionUnitAxisZ.commands.moveVelocity )
   END_RUNG
   // the same network as SCL:
   "Unit1.Em6.ControlNodes".cm.Interlock.visionUnit.source.moveVelocity := "Unit1.EmNodes".emRelations.em7.monitoring.cmStatus.cutConvAxis.statusWord1.Standstill;
   "Unit1.Em6.ControlNodes".cmVisionUnitAxisZ.commands.moveVelocity := NOT (NOT #FALSE);
END_REGION

REGION Network 49: CM Vision Z Axis Command stop
   RUNG wire#powerrail
      Contact( #TRUE )
      Coil( "Unit1.Em6.ControlNodes".cm.Interlock.visionUnit.source.stop )
   END_RUNG
   RUNG wire#powerrail
      I_Contact( #FALSE )
      Not()
      Coil( "Unit1.Em6.ControlNodes".cmVisionUnitAxisZ.commands.stop )
   END_RUNG
   // the same network as SCL:
   "Unit1.Em6.ControlNodes".cm.Interlock.visionUnit.source.stop := #TRUE;
   "Unit1.Em6.ControlNodes".cmVisionUnitAxisZ.commands.stop := NOT (NOT #FALSE);
END_REGION

REGION Network 50: CM Vision Z Axis Command fastStop
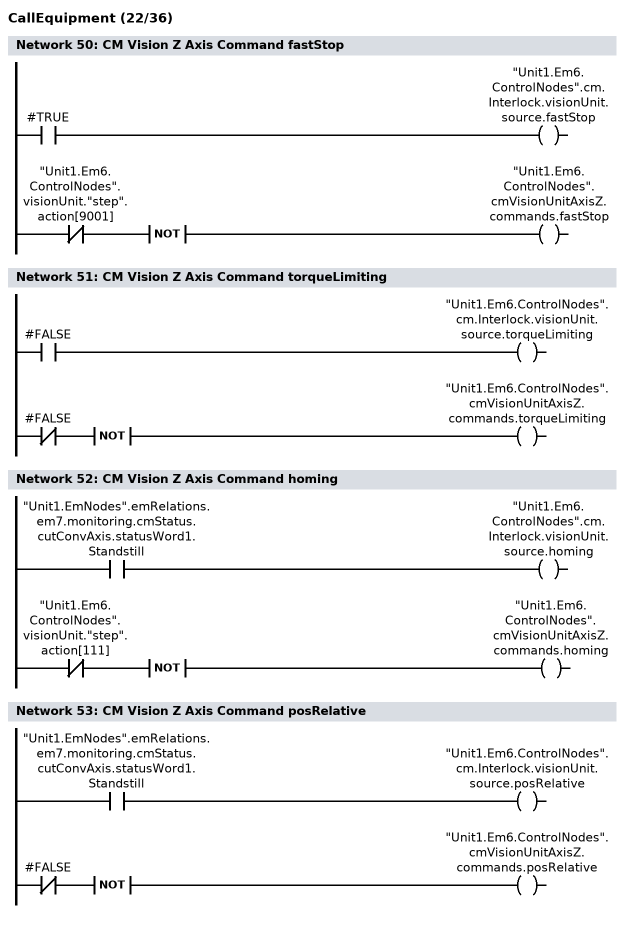
   RUNG wire#powerrail
      Contact( #TRUE )
      Coil( "Unit1.Em6.ControlNodes".cm.Interlock.visionUnit.source.fastStop )
   END_RUNG
   RUNG wire#powerrail
      I_Contact( "Unit1.Em6.ControlNodes".visionUnit."step".action[9001] )
      Not()
      Coil( "Unit1.Em6.ControlNodes".cmVisionUnitAxisZ.commands.fastStop )
   END_RUNG
   // the same network as SCL:
   "Unit1.Em6.ControlNodes".cm.Interlock.visionUnit.source.fastStop := #TRUE;
   "Unit1.Em6.ControlNodes".cmVisionUnitAxisZ.commands.fastStop := NOT (NOT "Unit1.Em6.ControlNodes".visionUnit."step".action[9001]);
END_REGION

REGION Network 51: CM Vision Z Axis Command torqueLimiting
   RUNG wire#powerrail
      Contact( #FALSE )
      Coil( "Unit1.Em6.ControlNodes".cm.Interlock.visionUnit.source.torqueLimiting )
   END_RUNG
   RUNG wire#powerrail
      I_Contact( #FALSE )
      Not()
      Coil( "Unit1.Em6.ControlNodes".cmVisionUnitAxisZ.commands.torqueLimiting )
   END_RUNG
   // the same network as SCL:
   "Unit1.Em6.ControlNodes".cm.Interlock.visionUnit.source.torqueLimiting := #FALSE;
   "Unit1.Em6.ControlNodes".cmVisionUnitAxisZ.commands.torqueLimiting := NOT (NOT #FALSE);
END_REGION

REGION Network 52: CM Vision Z Axis Command homing
   RUNG wire#powerrail
      Contact( "Unit1.EmNodes".emRelations.em7.monitoring.cmStatus.cutConvAxis.statusWord1.Standstill )
      Coil( "Unit1.Em6.ControlNodes".cm.Interlock.visionUnit.source.homing )
   END_RUNG
   RUNG wire#powerrail
      I_Contact( "Unit1.Em6.ControlNodes".visionUnit."step".action[111] )
      Not()
      Coil( "Unit1.Em6.ControlNodes".cmVisionUnitAxisZ.commands.homing )
   END_RUNG
   // the same network as SCL:
   "Unit1.Em6.ControlNodes".cm.Interlock.visionUnit.source.homing := "Unit1.EmNodes".emRelations.em7.monitoring.cmStatus.cutConvAxis.statusWord1.Standstill;
   "Unit1.Em6.ControlNodes".cmVisionUnitAxisZ.commands.homing := NOT (NOT "Unit1.Em6.ControlNodes".visionUnit."step".action[111]);
END_REGION

REGION Network 53: CM Vision Z Axis Command posRelative
   RUNG wire#powerrail
      Contact( "Unit1.EmNodes".emRelations.em7.monitoring.cmStatus.cutConvAxis.statusWord1.Standstill )
      Coil( "Unit1.Em6.ControlNodes".cm.Interlock.visionUnit.source.posRelative )
   END_RUNG
   RUNG wire#powerrail
      I_Contact( #FALSE )
      Not()
      Coil( "Unit1.Em6.ControlNodes".cmVisionUnitAxisZ.commands.posRelative )
   END_RUNG
   // the same network as SCL:
   "Unit1.Em6.ControlNodes".cm.Interlock.visionUnit.source.posRelative := "Unit1.EmNodes".emRelations.em7.monitoring.cmStatus.cutConvAxis.statusWord1.Standstill;
   "Unit1.Em6.ControlNodes".cmVisionUnitAxisZ.commands.posRelative := NOT (NOT #FALSE);
END_REGION

